// TIA Portal V16 export
// export: Created 2023-05-12T09:02:59.8974602Z, ExportSetting WithDefaults, DisplayName Totally Integrated Automation Portal, DisplayVersion V16 Update 3, DisplayName TIA Portal Version Control Interface, DisplayVersion V16 Update 2, DisplayName TIA Portal Openness, DisplayVersion V16 Update 3, DisplayName SINAMICS Startdrive Advanced, DisplayVersion V16, DisplayName SINAMICS Startdrive G130, G150, S120, S150, SINAMICS MV, S210, DisplayVersion V16, DisplayName SINAMICS Startdrive G110M, G120, G120C, G120D, G120P, DisplayVersion V16, DisplayName STEP 7 Professional, DisplayVersion V16 Update 3, DisplayName STEP 7 Safety, DisplayVersion V16, DisplayName WinCC Advanced, DisplayVersion V16 Update 3
FUNCTION "CIP_LINEA1" : Void   // FC53, LAD
{ S7_Optimized_Access := 'FALSE' }
VERSION : 0.1
// stored: AutoNumber false, IsIECCheckEnabled false, SetENOAutomatically false, UDAEnableTagReadback false
   VAR_TEMP
      AUX_TEM_P1 : S5Time;
      AUX_BOOL_1 : Bool;
   END_VAR
   VAR_TEMP   // added for the SCL form of the ladder/FBD networks
      _w1 : Bool;
      _s5time1 : S5Time;
   END_VAR
BEGIN

REGION Network 1: SOLO EN LIMPIEZA TANQUES
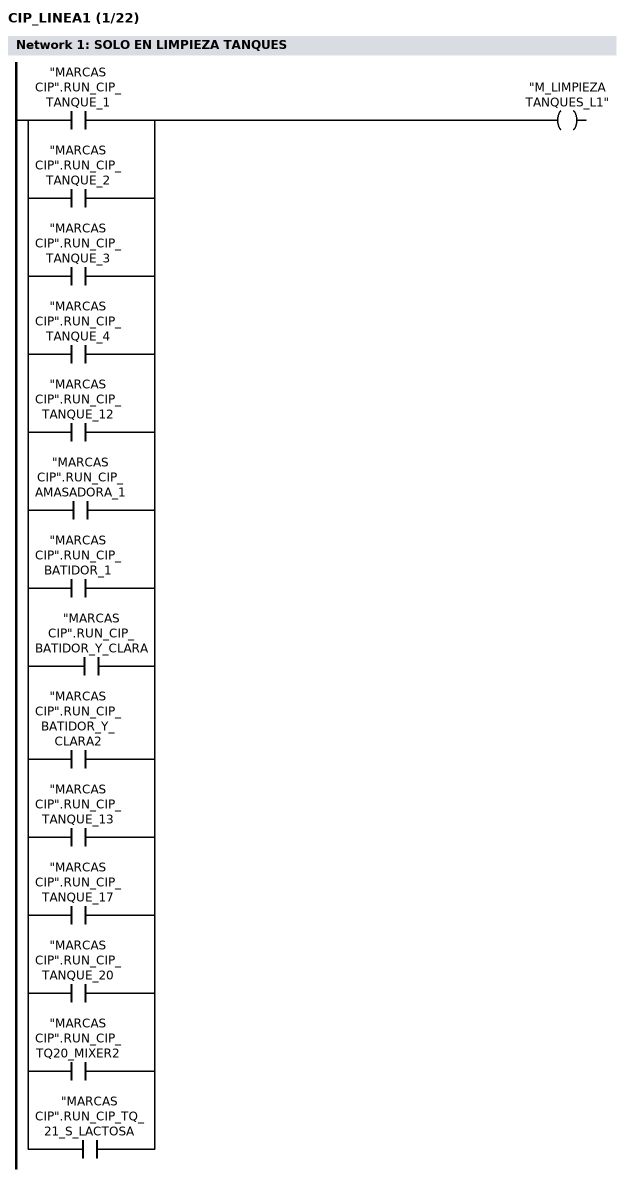
   RUNG wire#powerrail
      Contact( "MARCAS CIP".RUN_CIP_TANQUE_1 )
      wire#w1
      Coil( "M_LIMPIEZA TANQUES_L1" )
   END_RUNG
   RUNG wire#powerrail
      Contact( "MARCAS CIP".RUN_CIP_TANQUE_2 )
   END_RUNG wire#w1
   RUNG wire#powerrail
      Contact( "MARCAS CIP".RUN_CIP_TANQUE_3 )
   END_RUNG wire#w1
   RUNG wire#powerrail
      Contact( "MARCAS CIP".RUN_CIP_TANQUE_4 )
   END_RUNG wire#w1
   RUNG wire#powerrail
      Contact( "MARCAS CIP".RUN_CIP_TANQUE_12 )
   END_RUNG wire#w1
   RUNG wire#powerrail
      Contact( "MARCAS CIP".RUN_CIP_AMASADORA_1 )
   END_RUNG wire#w1
   RUNG wire#powerrail
      Contact( "MARCAS CIP".RUN_CIP_BATIDOR_1 )
   END_RUNG wire#w1
   RUNG wire#powerrail
      Contact( "MARCAS CIP".RUN_CIP_BATIDOR_Y_CLARA )
   END_RUNG wire#w1
   RUNG wire#powerrail
      Contact( "MARCAS CIP".RUN_CIP_BATIDOR_Y_CLARA2 )
   END_RUNG wire#w1
   RUNG wire#powerrail
      Contact( "MARCAS CIP".RUN_CIP_TANQUE_13 )
   END_RUNG wire#w1
   RUNG wire#powerrail
      Contact( "MARCAS CIP".RUN_CIP_TANQUE_17 )
   END_RUNG wire#w1
   RUNG wire#powerrail
      Contact( "MARCAS CIP".RUN_CIP_TANQUE_20 )
   END_RUNG wire#w1
   RUNG wire#powerrail
      Contact( "MARCAS CIP".RUN_CIP_TQ20_MIXER2 )
   END_RUNG wire#w1
   RUNG wire#powerrail
      Contact( "MARCAS CIP".RUN_CIP_TQ_21_S_LACTOSA )
   END_RUNG wire#w1
   // the same network as SCL:
   "M_LIMPIEZA TANQUES_L1" := "MARCAS CIP".RUN_CIP_TANQUE_1 OR "MARCAS CIP".RUN_CIP_TANQUE_2 OR "MARCAS CIP".RUN_CIP_TANQUE_3 OR "MARCAS CIP".RUN_CIP_TANQUE_4 OR "MARCAS CIP".RUN_CIP_TANQUE_12 OR "MARCAS CIP".RUN_CIP_AMASADORA_1 OR "MARCAS CIP".RUN_CIP_BATIDOR_1 OR "MARCAS CIP".RUN_CIP_BATIDOR_Y_CLARA OR "MARCAS CIP".RUN_CIP_BATIDOR_Y_CLARA2 OR "MARCAS CIP".RUN_CIP_TANQUE_13 OR "MARCAS CIP".RUN_CIP_TANQUE_17 OR "MARCAS CIP".RUN_CIP_TANQUE_20 OR "MARCAS CIP".RUN_CIP_TQ20_MIXER2 OR "MARCAS CIP".RUN_CIP_TQ_21_S_LACTOSA;
END_REGION

REGION Network 2: PASO 1 PRIEMER ENJUEGE AGUA RECUPERADA
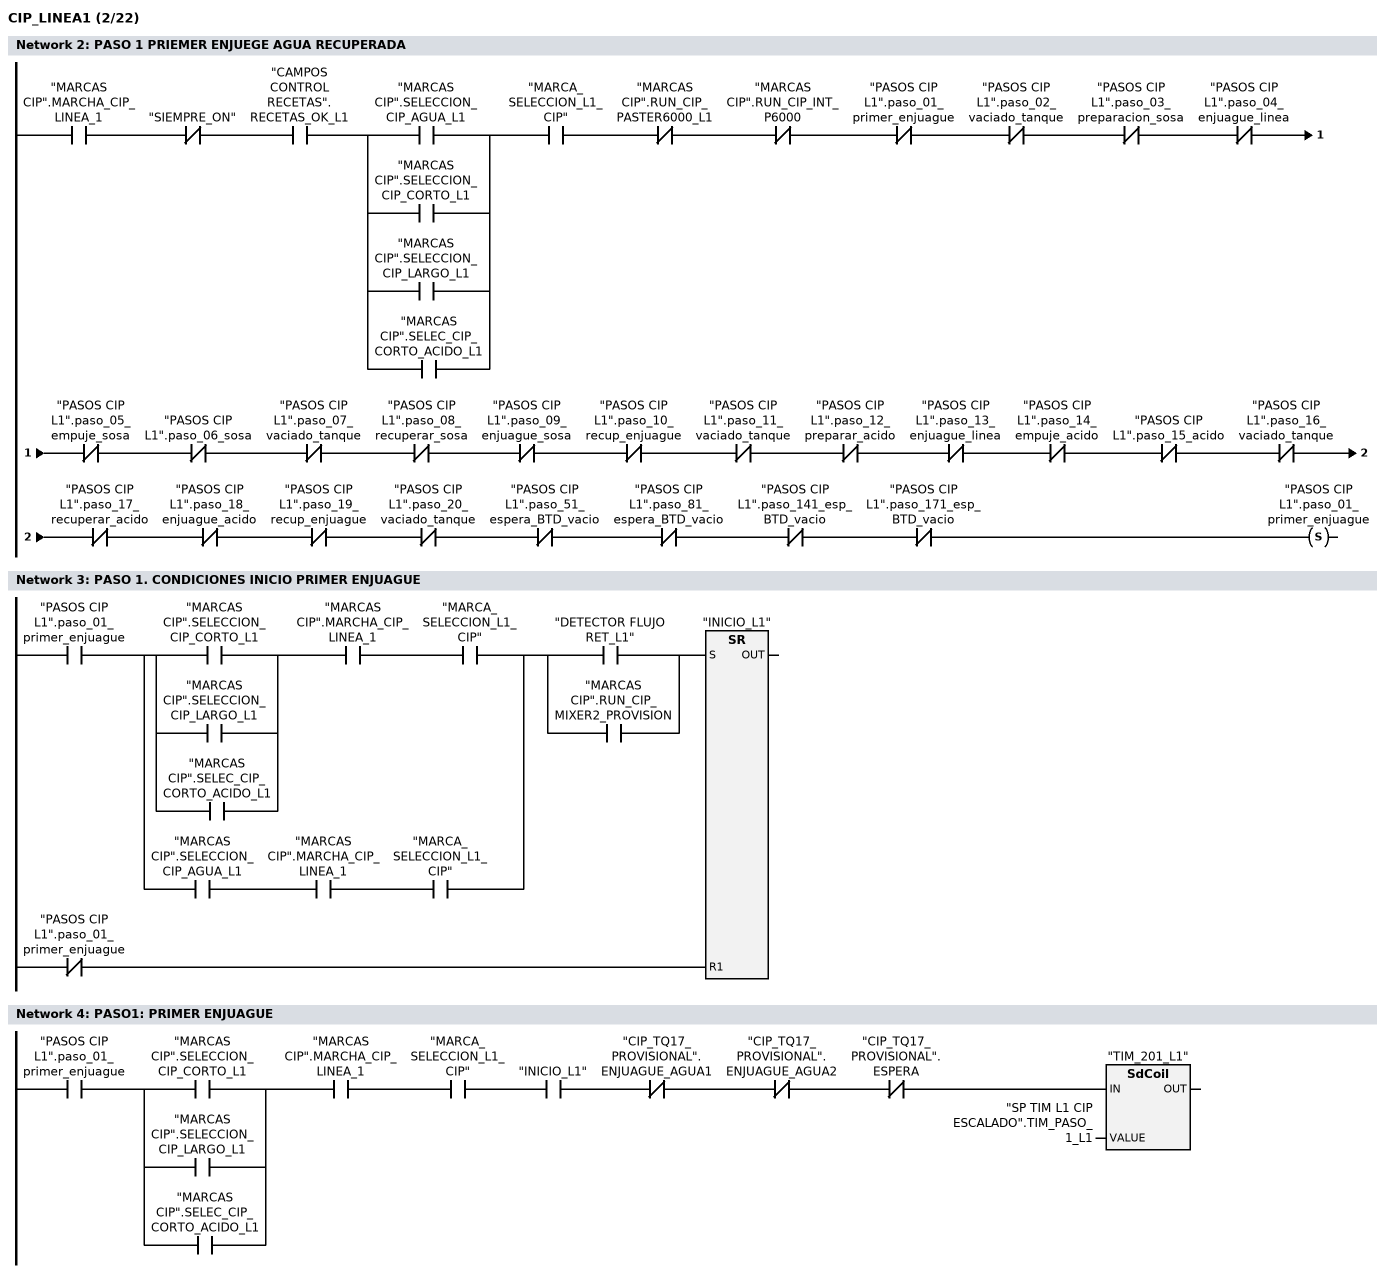
   RUNG wire#powerrail
      Contact( "MARCAS CIP".MARCHA_CIP_LINEA_1 )
      I_Contact( "SIEMPRE_ON" )
      Contact( "CAMPOS CONTROL RECETAS".RECETAS_OK_L1 )
      wire#w1
      Contact( "MARCAS CIP".SELECCION_CIP_AGUA_L1 )
      wire#w2
      Contact( "MARCA_SELECCION_L1_CIP" )
      I_Contact( "MARCAS CIP".RUN_CIP_PASTER6000_L1 )
      I_Contact( "MARCAS CIP".RUN_CIP_INT_P6000 )
      I_Contact( "PASOS CIP L1".paso_01_primer_enjuague )
      I_Contact( "PASOS CIP L1".paso_02_vaciado_tanque )
      I_Contact( "PASOS CIP L1".paso_03_preparacion_sosa )
      I_Contact( "PASOS CIP L1".paso_04_enjuague_linea )
      I_Contact( "PASOS CIP L1".paso_05_empuje_sosa )
      I_Contact( "PASOS CIP L1".paso_06_sosa )
      I_Contact( "PASOS CIP L1".paso_07_vaciado_tanque )
      I_Contact( "PASOS CIP L1".paso_08_recuperar_sosa )
      I_Contact( "PASOS CIP L1".paso_09_enjuague_sosa )
      I_Contact( "PASOS CIP L1".paso_10_recup_enjuague )
      I_Contact( "PASOS CIP L1".paso_11_vaciado_tanque )
      I_Contact( "PASOS CIP L1".paso_12_preparar_acido )
      I_Contact( "PASOS CIP L1".paso_13_enjuague_linea )
      I_Contact( "PASOS CIP L1".paso_14_empuje_acido )
      I_Contact( "PASOS CIP L1".paso_15_acido )
      I_Contact( "PASOS CIP L1".paso_16_vaciado_tanque )
      I_Contact( "PASOS CIP L1".paso_17_recuperar_acido )
      I_Contact( "PASOS CIP L1".paso_18_enjuague_acido )
      I_Contact( "PASOS CIP L1".paso_19_recup_enjuague )
      I_Contact( "PASOS CIP L1".paso_20_vaciado_tanque )
      I_Contact( "PASOS CIP L1".paso_51_espera_BTD_vacio )
      I_Contact( "PASOS CIP L1".paso_81_espera_BTD_vacio )
      I_Contact( "PASOS CIP L1".paso_141_esp_BTD_vacio )
      I_Contact( "PASOS CIP L1".paso_171_esp_BTD_vacio )
      S_Coil( "PASOS CIP L1".paso_01_primer_enjuague )
   END_RUNG
   RUNG wire#w1
      Contact( "MARCAS CIP".SELECCION_CIP_CORTO_L1 )
   END_RUNG wire#w2
   RUNG wire#w1
      Contact( "MARCAS CIP".SELECCION_CIP_LARGO_L1 )
   END_RUNG wire#w2
   RUNG wire#w1
      Contact( "MARCAS CIP".SELEC_CIP_CORTO_ACIDO_L1 )
   END_RUNG wire#w2
   // the same network as SCL:
   IF "MARCAS CIP".MARCHA_CIP_LINEA_1 AND NOT "SIEMPRE_ON" AND "CAMPOS CONTROL RECETAS".RECETAS_OK_L1 AND ("MARCAS CIP".SELECCION_CIP_AGUA_L1 OR "MARCAS CIP".SELECCION_CIP_CORTO_L1 OR "MARCAS CIP".SELECCION_CIP_LARGO_L1 OR "MARCAS CIP".SELEC_CIP_CORTO_ACIDO_L1) AND "MARCA_SELECCION_L1_CIP" AND NOT "MARCAS CIP".RUN_CIP_PASTER6000_L1 AND NOT "MARCAS CIP".RUN_CIP_INT_P6000 AND NOT "PASOS CIP L1".paso_01_primer_enjuague AND NOT "PASOS CIP L1".paso_02_vaciado_tanque AND NOT "PASOS CIP L1".paso_03_preparacion_sosa AND NOT "PASOS CIP L1".paso_04_enjuague_linea AND NOT "PASOS CIP L1".paso_05_empuje_sosa AND NOT "PASOS CIP L1".paso_06_sosa AND NOT "PASOS CIP L1".paso_07_vaciado_tanque AND NOT "PASOS CIP L1".paso_08_recuperar_sosa AND NOT "PASOS CIP L1".paso_09_enjuague_sosa AND NOT "PASOS CIP L1".paso_10_recup_enjuague AND NOT "PASOS CIP L1".paso_11_vaciado_tanque AND NOT "PASOS CIP L1".paso_12_preparar_acido AND NOT "PASOS CIP L1".paso_13_enjuague_linea AND NOT "PASOS CIP L1".paso_14_empuje_acido AND NOT "PASOS CIP L1".paso_15_acido AND NOT "PASOS CIP L1".paso_16_vaciado_tanque AND NOT "PASOS CIP L1".paso_17_recuperar_acido AND NOT "PASOS CIP L1".paso_18_enjuague_acido AND NOT "PASOS CIP L1".paso_19_recup_enjuague AND NOT "PASOS CIP L1".paso_20_vaciado_tanque AND NOT "PASOS CIP L1".paso_51_espera_BTD_vacio AND NOT "PASOS CIP L1".paso_81_espera_BTD_vacio AND NOT "PASOS CIP L1".paso_141_esp_BTD_vacio AND NOT "PASOS CIP L1".paso_171_esp_BTD_vacio THEN
       "PASOS CIP L1".paso_01_primer_enjuague := TRUE;
   END_IF;
END_REGION

REGION Network 3: PASO 1. CONDICIONES INICIO PRIMER ENJUAGUE
   RUNG wire#powerrail
      Contact( "PASOS CIP L1".paso_01_primer_enjuague )
      wire#w1
      Contact( "MARCAS CIP".SELECCION_CIP_CORTO_L1 )
      wire#w2
      Contact( "MARCAS CIP".MARCHA_CIP_LINEA_1 )
      Contact( "MARCA_SELECCION_L1_CIP" )
      wire#w3
      Contact( "DETECTOR FLUJO RET_L1" )
      wire#w4
      S_SR(operand := "INICIO_L1", r1 := wire#w5)
   END_RUNG
   RUNG wire#w1
      Contact( "MARCAS CIP".SELECCION_CIP_LARGO_L1 )
   END_RUNG wire#w2
   RUNG wire#w1
      Contact( "MARCAS CIP".SELEC_CIP_CORTO_ACIDO_L1 )
   END_RUNG wire#w2
   RUNG wire#w1
      Contact( "MARCAS CIP".SELECCION_CIP_AGUA_L1 )
      Contact( "MARCAS CIP".MARCHA_CIP_LINEA_1 )
      Contact( "MARCA_SELECCION_L1_CIP" )
   END_RUNG wire#w3
   RUNG wire#w3
      Contact( "MARCAS CIP".RUN_CIP_MIXER2_PROVISION )
   END_RUNG wire#w4
   RUNG wire#powerrail
      I_Contact( "PASOS CIP L1".paso_01_primer_enjuague )
   END_RUNG wire#w5
   // the same network as SCL:
   IF "PASOS CIP L1".paso_01_primer_enjuague AND ((("MARCAS CIP".SELECCION_CIP_CORTO_L1 OR "MARCAS CIP".SELECCION_CIP_LARGO_L1 OR "MARCAS CIP".SELEC_CIP_CORTO_ACIDO_L1) AND "MARCAS CIP".MARCHA_CIP_LINEA_1 AND "MARCA_SELECCION_L1_CIP") OR ("MARCAS CIP".SELECCION_CIP_AGUA_L1 AND "MARCAS CIP".MARCHA_CIP_LINEA_1 AND "MARCA_SELECCION_L1_CIP")) AND ("DETECTOR FLUJO RET_L1" OR "MARCAS CIP".RUN_CIP_MIXER2_PROVISION) THEN
       "INICIO_L1" := TRUE;   // SR flip-flop
   END_IF;
   IF NOT "PASOS CIP L1".paso_01_primer_enjuague THEN "INICIO_L1" := FALSE; END_IF;
END_REGION

REGION Network 4: PASO1: PRIMER ENJUAGUE
   // no SCL statement known for SdCoil: written as a call
   SdCoil(value := "SP TIM L1 CIP ESCALADO".TIM_PASO_1_L1,
          operand := "TIM_201_L1",
          in := "PASOS CIP L1".paso_01_primer_enjuague AND ("MARCAS CIP".SELECCION_CIP_CORTO_L1 OR "MARCAS CIP".SELECCION_CIP_LARGO_L1 OR "MARCAS CIP".SELEC_CIP_CORTO_ACIDO_L1) AND "MARCAS CIP".MARCHA_CIP_LINEA_1 AND "MARCA_SELECCION_L1_CIP" AND "INICIO_L1" AND NOT "CIP_TQ17_PROVISIONAL".ENJUAGUE_AGUA1 AND NOT "CIP_TQ17_PROVISIONAL".ENJUAGUE_AGUA2 AND NOT "CIP_TQ17_PROVISIONAL".ESPERA);
END_REGION

REGION Network 5: PASO 2: VACIADO TANQUE (SOLO BOMBA RETORNO CIP)
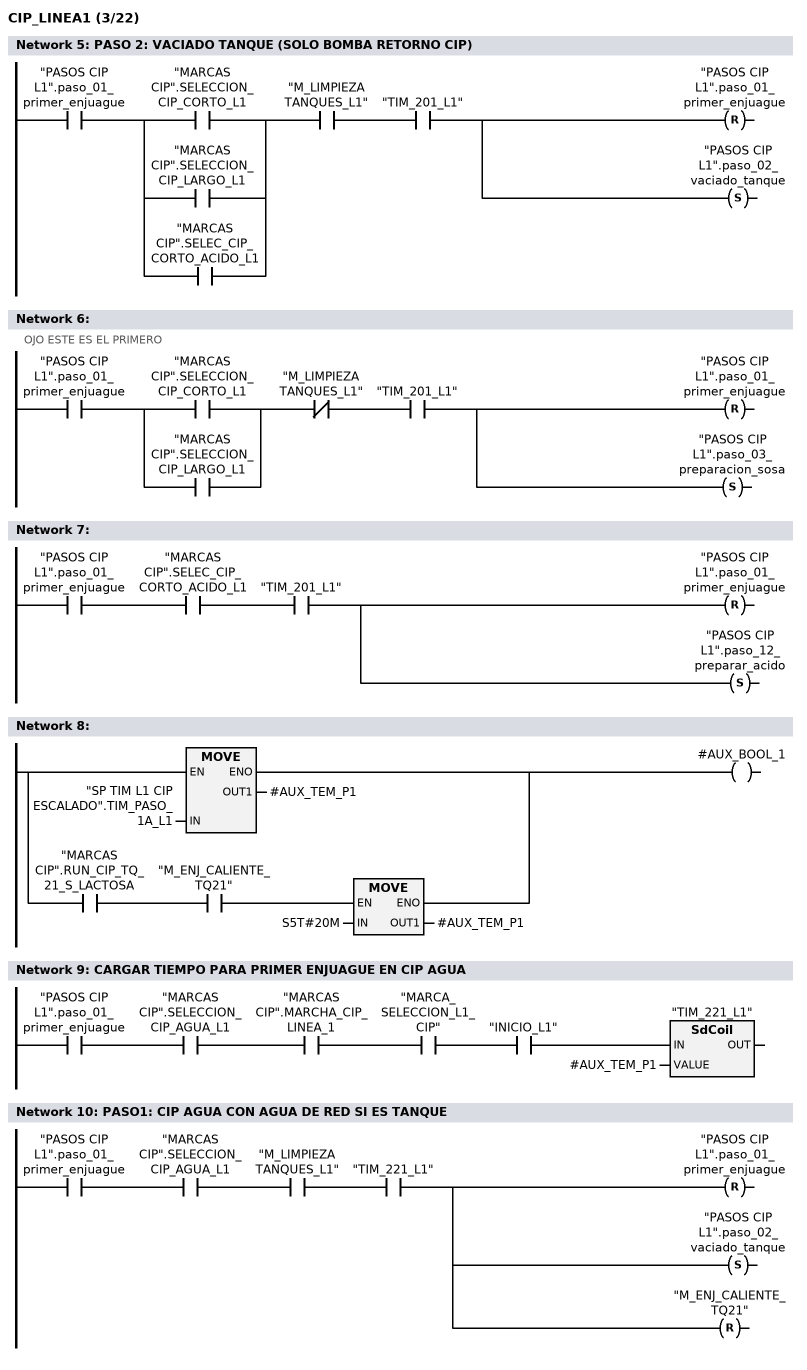
   RUNG wire#powerrail
      Contact( "PASOS CIP L1".paso_01_primer_enjuague )
      wire#w1
      Contact( "MARCAS CIP".SELECCION_CIP_CORTO_L1 )
      wire#w2
      Contact( "M_LIMPIEZA TANQUES_L1" )
      Contact( "TIM_201_L1" )
      wire#w3
      R_Coil( "PASOS CIP L1".paso_01_primer_enjuague )
   END_RUNG
   RUNG wire#w1
      Contact( "MARCAS CIP".SELECCION_CIP_LARGO_L1 )
   END_RUNG wire#w2
   RUNG wire#w1
      Contact( "MARCAS CIP".SELEC_CIP_CORTO_ACIDO_L1 )
   END_RUNG wire#w2
   RUNG wire#w3
      S_Coil( "PASOS CIP L1".paso_02_vaciado_tanque )
   END_RUNG
   // the same network as SCL:
   #_w1 := "PASOS CIP L1".paso_01_primer_enjuague AND ("MARCAS CIP".SELECCION_CIP_CORTO_L1 OR "MARCAS CIP".SELECCION_CIP_LARGO_L1 OR "MARCAS CIP".SELEC_CIP_CORTO_ACIDO_L1) AND "M_LIMPIEZA TANQUES_L1" AND "TIM_201_L1";
   IF #_w1 THEN
       "PASOS CIP L1".paso_01_primer_enjuague := FALSE;
       "PASOS CIP L1".paso_02_vaciado_tanque := TRUE;
   END_IF;
END_REGION

REGION Network 6
   // OJO ESTE ES EL PRIMERO
   RUNG wire#powerrail
      Contact( "PASOS CIP L1".paso_01_primer_enjuague )
      wire#w1
      Contact( "MARCAS CIP".SELECCION_CIP_CORTO_L1 )
      wire#w2
      I_Contact( "M_LIMPIEZA TANQUES_L1" )
      Contact( "TIM_201_L1" )
      wire#w3
      R_Coil( "PASOS CIP L1".paso_01_primer_enjuague )
   END_RUNG
   RUNG wire#w1
      Contact( "MARCAS CIP".SELECCION_CIP_LARGO_L1 )
   END_RUNG wire#w2
   RUNG wire#w3
      S_Coil( "PASOS CIP L1".paso_03_preparacion_sosa )
   END_RUNG
   // the same network as SCL:
   #_w1 := "PASOS CIP L1".paso_01_primer_enjuague AND ("MARCAS CIP".SELECCION_CIP_CORTO_L1 OR "MARCAS CIP".SELECCION_CIP_LARGO_L1) AND NOT "M_LIMPIEZA TANQUES_L1" AND "TIM_201_L1";
   IF #_w1 THEN
       "PASOS CIP L1".paso_01_primer_enjuague := FALSE;
       "PASOS CIP L1".paso_03_preparacion_sosa := TRUE;
   END_IF;
END_REGION

REGION Network 7
   RUNG wire#powerrail
      Contact( "PASOS CIP L1".paso_01_primer_enjuague )
      Contact( "MARCAS CIP".SELEC_CIP_CORTO_ACIDO_L1 )
      Contact( "TIM_201_L1" )
      wire#w1
      R_Coil( "PASOS CIP L1".paso_01_primer_enjuague )
   END_RUNG
   RUNG wire#w1
      S_Coil( "PASOS CIP L1".paso_12_preparar_acido )
   END_RUNG
   // the same network as SCL:
   #_w1 := "PASOS CIP L1".paso_01_primer_enjuague AND "MARCAS CIP".SELEC_CIP_CORTO_ACIDO_L1 AND "TIM_201_L1";
   IF #_w1 THEN
       "PASOS CIP L1".paso_01_primer_enjuague := FALSE;
       "PASOS CIP L1".paso_12_preparar_acido := TRUE;
   END_IF;
END_REGION

REGION Network 8
   RUNG wire#powerrail
      { S7_GenerateENO := "TRUE" } Move(in := "SP TIM L1 CIP ESCALADO".TIM_PASO_1A_L1, out1 => #AUX_TEM_P1)
      wire#w1
      Coil( #AUX_BOOL_1 )
   END_RUNG
   RUNG wire#powerrail
      Contact( "MARCAS CIP".RUN_CIP_TQ_21_S_LACTOSA )
      Contact( "M_ENJ_CALIENTE_TQ21" )
      { S7_GenerateENO := "TRUE" } Move(in := S5T#20M, out1 => #AUX_TEM_P1)
   END_RUNG wire#w1
   // the same network as SCL:
   // ENO of a box is taken as its EN; it also drops when the box reports an error
   #AUX_TEM_P1 := "SP TIM L1 CIP ESCALADO".TIM_PASO_1A_L1;
   #_w1 := "MARCAS CIP".RUN_CIP_TQ_21_S_LACTOSA AND "M_ENJ_CALIENTE_TQ21";
   IF #_w1 THEN #AUX_TEM_P1 := S5T#20M; END_IF;
   #AUX_BOOL_1 := TRUE OR #_w1;
END_REGION

REGION Network 9: CARGAR TIEMPO PARA PRIMER ENJUAGUE EN CIP AGUA
   // no SCL statement known for SdCoil: written as a call
   SdCoil(value := #AUX_TEM_P1,
          operand := "TIM_221_L1",
          in := "PASOS CIP L1".paso_01_primer_enjuague AND "MARCAS CIP".SELECCION_CIP_AGUA_L1 AND "MARCAS CIP".MARCHA_CIP_LINEA_1 AND "MARCA_SELECCION_L1_CIP" AND "INICIO_L1");
END_REGION

REGION Network 10: PASO1: CIP AGUA CON AGUA DE RED SI ES TANQUE
   RUNG wire#powerrail
      Contact( "PASOS CIP L1".paso_01_primer_enjuague )
      Contact( "MARCAS CIP".SELECCION_CIP_AGUA_L1 )
      Contact( "M_LIMPIEZA TANQUES_L1" )
      Contact( "TIM_221_L1" )
      wire#w1
      R_Coil( "PASOS CIP L1".paso_01_primer_enjuague )
   END_RUNG
   RUNG wire#w1
      S_Coil( "PASOS CIP L1".paso_02_vaciado_tanque )
   END_RUNG
   RUNG wire#w1
      R_Coil( "M_ENJ_CALIENTE_TQ21" )
   END_RUNG
   // the same network as SCL:
   #_w1 := "PASOS CIP L1".paso_01_primer_enjuague AND "MARCAS CIP".SELECCION_CIP_AGUA_L1 AND "M_LIMPIEZA TANQUES_L1" AND "TIM_221_L1";
   IF #_w1 THEN
       "PASOS CIP L1".paso_01_primer_enjuague := FALSE;
       "PASOS CIP L1".paso_02_vaciado_tanque := TRUE;
       "M_ENJ_CALIENTE_TQ21" := FALSE;
   END_IF;
END_REGION

REGION Network 11: PASO1: CIP AGUA CON AGUA DE RED SI ES LINEA
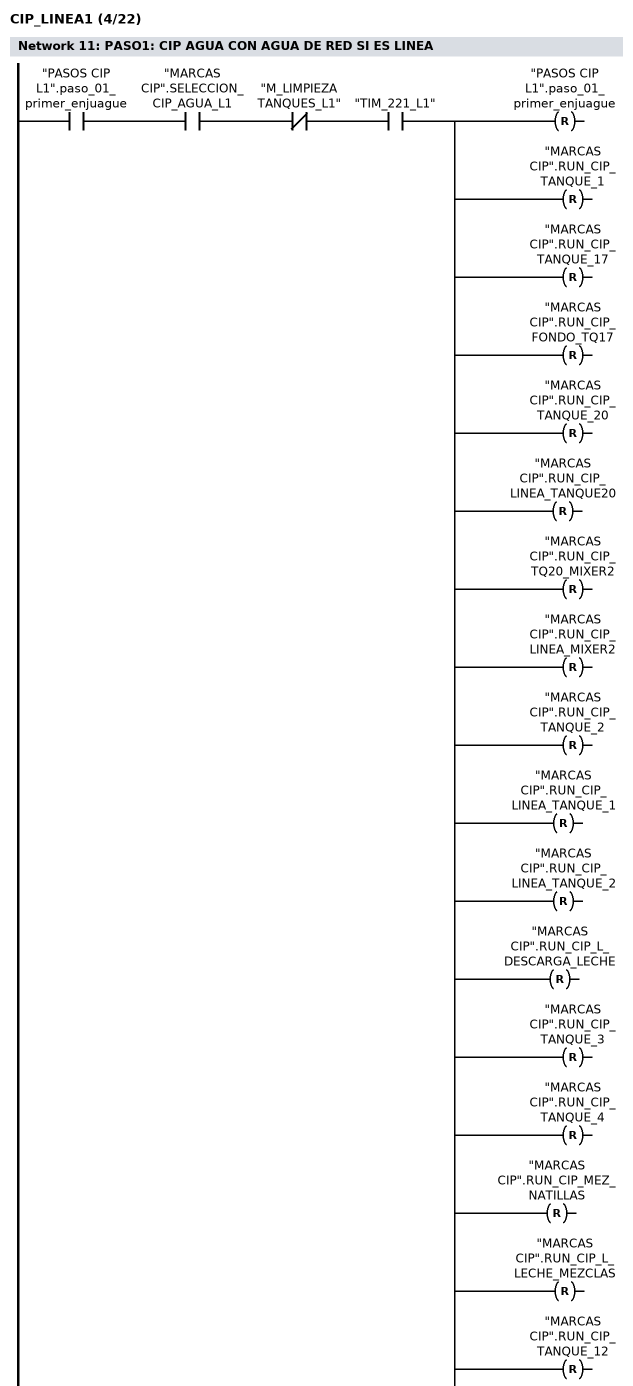
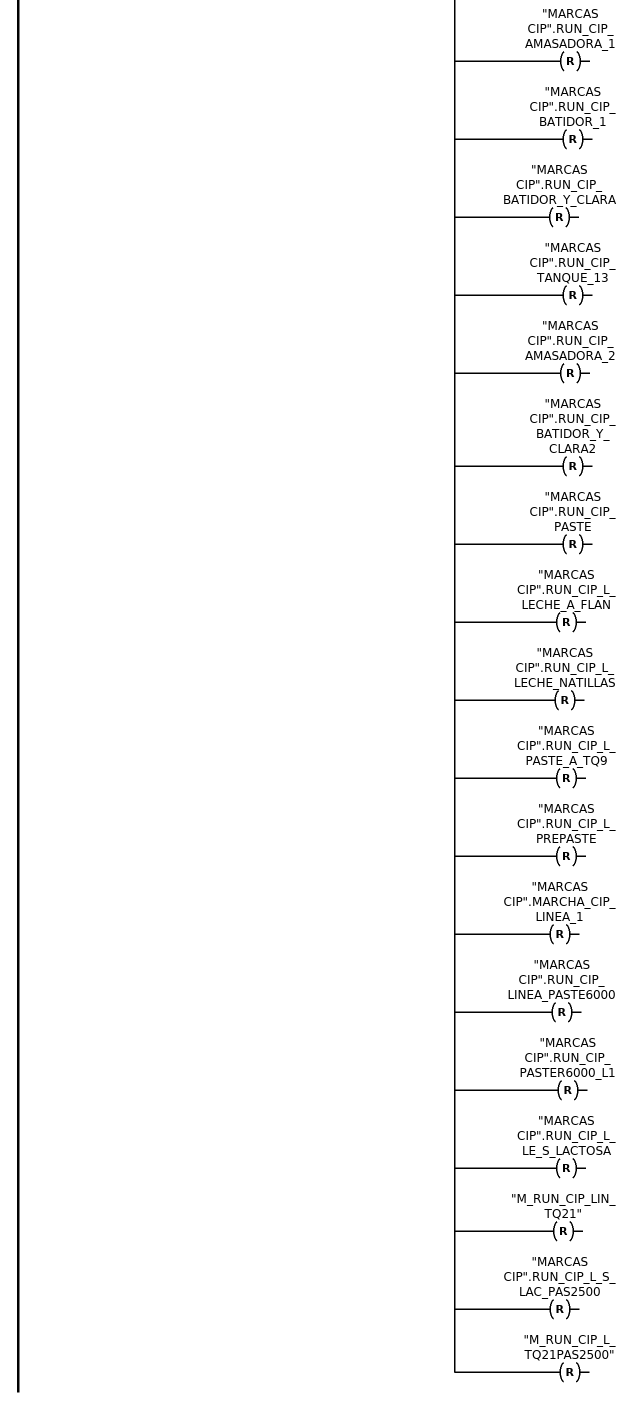
   RUNG wire#powerrail
      Contact( "PASOS CIP L1".paso_01_primer_enjuague )
      Contact( "MARCAS CIP".SELECCION_CIP_AGUA_L1 )
      I_Contact( "M_LIMPIEZA TANQUES_L1" )
      Contact( "TIM_221_L1" )
      wire#w1
      R_Coil( "PASOS CIP L1".paso_01_primer_enjuague )
   END_RUNG
   RUNG wire#w1
      R_Coil( "MARCAS CIP".RUN_CIP_TANQUE_1 )
   END_RUNG
   RUNG wire#w1
      R_Coil( "MARCAS CIP".RUN_CIP_TANQUE_17 )
   END_RUNG
   RUNG wire#w1
      R_Coil( "MARCAS CIP".RUN_CIP_FONDO_TQ17 )
   END_RUNG
   RUNG wire#w1
      R_Coil( "MARCAS CIP".RUN_CIP_TANQUE_20 )
   END_RUNG
   RUNG wire#w1
      R_Coil( "MARCAS CIP".RUN_CIP_LINEA_TANQUE20 )
   END_RUNG
   RUNG wire#w1
      R_Coil( "MARCAS CIP".RUN_CIP_TQ20_MIXER2 )
   END_RUNG
   RUNG wire#w1
      R_Coil( "MARCAS CIP".RUN_CIP_LINEA_MIXER2 )
   END_RUNG
   RUNG wire#w1
      R_Coil( "MARCAS CIP".RUN_CIP_TANQUE_2 )
   END_RUNG
   RUNG wire#w1
      R_Coil( "MARCAS CIP".RUN_CIP_LINEA_TANQUE_1 )
   END_RUNG
   RUNG wire#w1
      R_Coil( "MARCAS CIP".RUN_CIP_LINEA_TANQUE_2 )
   END_RUNG
   RUNG wire#w1
      R_Coil( "MARCAS CIP".RUN_CIP_L_DESCARGA_LECHE )
   END_RUNG
   RUNG wire#w1
      R_Coil( "MARCAS CIP".RUN_CIP_TANQUE_3 )
   END_RUNG
   RUNG wire#w1
      R_Coil( "MARCAS CIP".RUN_CIP_TANQUE_4 )
   END_RUNG
   RUNG wire#w1
      R_Coil( "MARCAS CIP".RUN_CIP_MEZ_NATILLAS )
   END_RUNG
   RUNG wire#w1
      R_Coil( "MARCAS CIP".RUN_CIP_L_LECHE_MEZCLAS )
   END_RUNG
   RUNG wire#w1
      R_Coil( "MARCAS CIP".RUN_CIP_TANQUE_12 )
   END_RUNG
   RUNG wire#w1
      R_Coil( "MARCAS CIP".RUN_CIP_AMASADORA_1 )
   END_RUNG
   RUNG wire#w1
      R_Coil( "MARCAS CIP".RUN_CIP_BATIDOR_1 )
   END_RUNG
   RUNG wire#w1
      R_Coil( "MARCAS CIP".RUN_CIP_BATIDOR_Y_CLARA )
   END_RUNG
   RUNG wire#w1
      R_Coil( "MARCAS CIP".RUN_CIP_TANQUE_13 )
   END_RUNG
   RUNG wire#w1
      R_Coil( "MARCAS CIP".RUN_CIP_AMASADORA_2 )
   END_RUNG
   RUNG wire#w1
      R_Coil( "MARCAS CIP".RUN_CIP_BATIDOR_Y_CLARA2 )
   END_RUNG
   RUNG wire#w1
      R_Coil( "MARCAS CIP".RUN_CIP_PASTE )
   END_RUNG
   RUNG wire#w1
      R_Coil( "MARCAS CIP".RUN_CIP_L_LECHE_A_FLAN )
   END_RUNG
   RUNG wire#w1
      R_Coil( "MARCAS CIP".RUN_CIP_L_LECHE_NATILLAS )
   END_RUNG
   RUNG wire#w1
      R_Coil( "MARCAS CIP".RUN_CIP_L_PASTE_A_TQ9 )
   END_RUNG
   RUNG wire#w1
      R_Coil( "MARCAS CIP".RUN_CIP_L_PREPASTE )
   END_RUNG
   RUNG wire#w1
      R_Coil( "MARCAS CIP".MARCHA_CIP_LINEA_1 )
   END_RUNG
   RUNG wire#w1
      R_Coil( "MARCAS CIP".RUN_CIP_LINEA_PASTE6000 )
   END_RUNG
   RUNG wire#w1
      R_Coil( "MARCAS CIP".RUN_CIP_PASTER6000_L1 )
   END_RUNG
   RUNG wire#w1
      R_Coil( "MARCAS CIP".RUN_CIP_L_LE_S_LACTOSA )
   END_RUNG
   RUNG wire#w1
      R_Coil( "M_RUN_CIP_LIN_TQ21" )
   END_RUNG
   RUNG wire#w1
      R_Coil( "MARCAS CIP".RUN_CIP_L_S_LAC_PAS2500 )
   END_RUNG
   RUNG wire#w1
      R_Coil( "M_RUN_CIP_L_TQ21PAS2500" )
   END_RUNG
   // the same network as SCL:
   #_w1 := "PASOS CIP L1".paso_01_primer_enjuague AND "MARCAS CIP".SELECCION_CIP_AGUA_L1 AND NOT "M_LIMPIEZA TANQUES_L1" AND "TIM_221_L1";
   IF #_w1 THEN
       "PASOS CIP L1".paso_01_primer_enjuague := FALSE;
       "MARCAS CIP".RUN_CIP_TANQUE_1 := FALSE;
       "MARCAS CIP".RUN_CIP_TANQUE_17 := FALSE;
       "MARCAS CIP".RUN_CIP_FONDO_TQ17 := FALSE;
       "MARCAS CIP".RUN_CIP_TANQUE_20 := FALSE;
       "MARCAS CIP".RUN_CIP_LINEA_TANQUE20 := FALSE;
       "MARCAS CIP".RUN_CIP_TQ20_MIXER2 := FALSE;
       "MARCAS CIP".RUN_CIP_LINEA_MIXER2 := FALSE;
       "MARCAS CIP".RUN_CIP_TANQUE_2 := FALSE;
       "MARCAS CIP".RUN_CIP_LINEA_TANQUE_1 := FALSE;
       "MARCAS CIP".RUN_CIP_LINEA_TANQUE_2 := FALSE;
       "MARCAS CIP".RUN_CIP_L_DESCARGA_LECHE := FALSE;
       "MARCAS CIP".RUN_CIP_TANQUE_3 := FALSE;
       "MARCAS CIP".RUN_CIP_TANQUE_4 := FALSE;
       "MARCAS CIP".RUN_CIP_MEZ_NATILLAS := FALSE;
       "MARCAS CIP".RUN_CIP_L_LECHE_MEZCLAS := FALSE;
       "MARCAS CIP".RUN_CIP_TANQUE_12 := FALSE;
       "MARCAS CIP".RUN_CIP_AMASADORA_1 := FALSE;
       "MARCAS CIP".RUN_CIP_BATIDOR_1 := FALSE;
       "MARCAS CIP".RUN_CIP_BATIDOR_Y_CLARA := FALSE;
       "MARCAS CIP".RUN_CIP_TANQUE_13 := FALSE;
       "MARCAS CIP".RUN_CIP_AMASADORA_2 := FALSE;
       "MARCAS CIP".RUN_CIP_BATIDOR_Y_CLARA2 := FALSE;
       "MARCAS CIP".RUN_CIP_PASTE := FALSE;
       "MARCAS CIP".RUN_CIP_L_LECHE_A_FLAN := FALSE;
       "MARCAS CIP".RUN_CIP_L_LECHE_NATILLAS := FALSE;
       "MARCAS CIP".RUN_CIP_L_PASTE_A_TQ9 := FALSE;
       "MARCAS CIP".RUN_CIP_L_PREPASTE := FALSE;
       "MARCAS CIP".MARCHA_CIP_LINEA_1 := FALSE;
       "MARCAS CIP".RUN_CIP_LINEA_PASTE6000 := FALSE;
       "MARCAS CIP".RUN_CIP_PASTER6000_L1 := FALSE;
       "MARCAS CIP".RUN_CIP_L_LE_S_LACTOSA := FALSE;
       "M_RUN_CIP_LIN_TQ21" := FALSE;
       "MARCAS CIP".RUN_CIP_L_S_LAC_PAS2500 := FALSE;
       "M_RUN_CIP_L_TQ21PAS2500" := FALSE;
   END_IF;
END_REGION

REGION Network 12
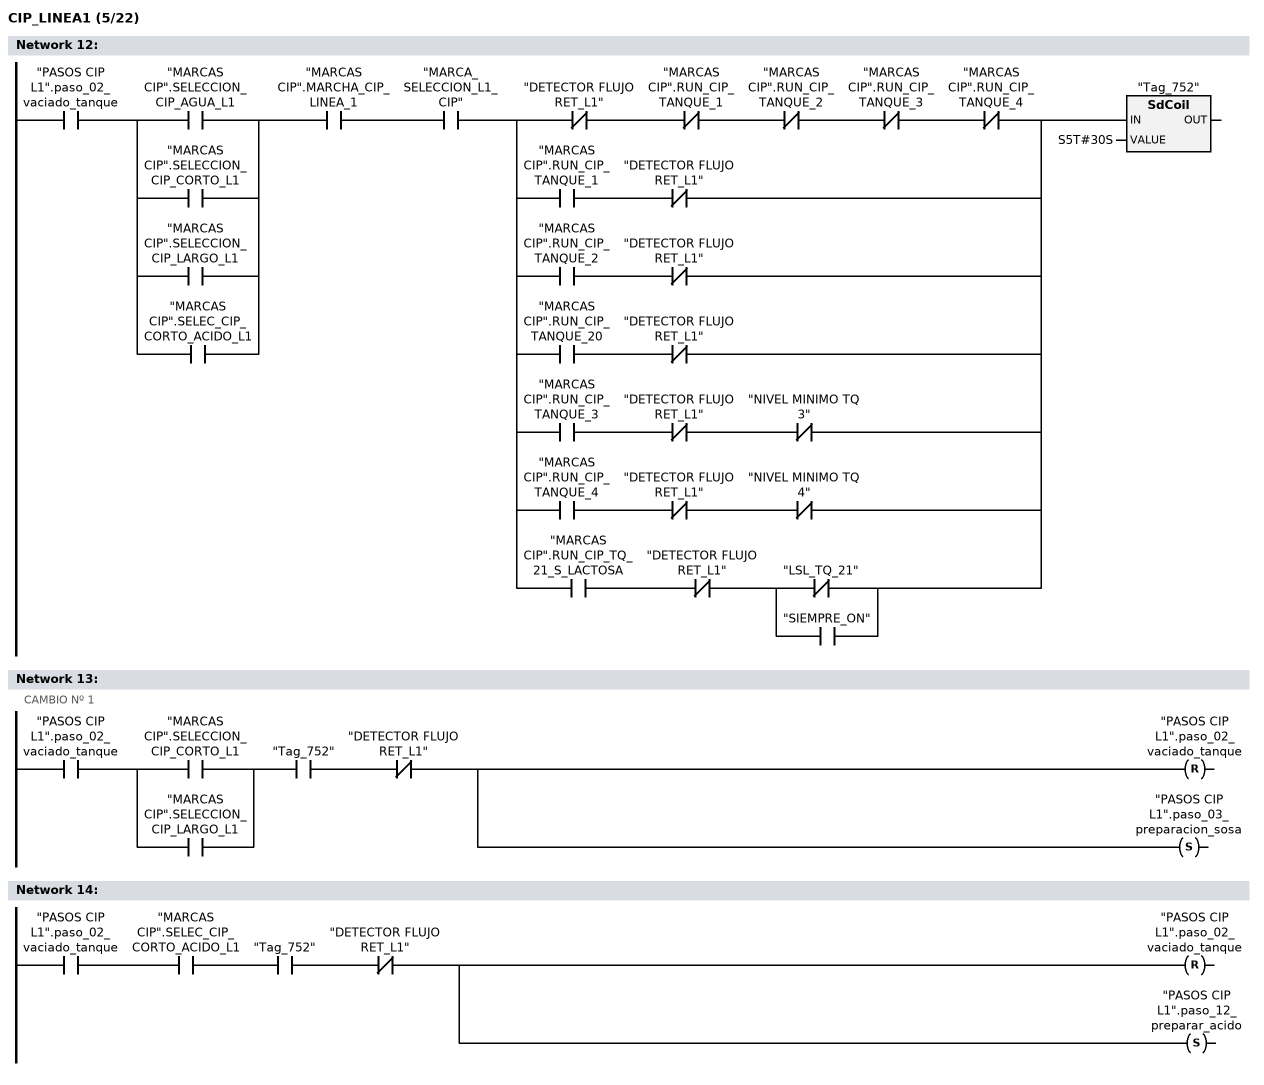
   // no SCL statement known for SdCoil: written as a call
   SdCoil(value := S5T#30S,
          in := "PASOS CIP L1".paso_02_vaciado_tanque AND ("MARCAS CIP".SELECCION_CIP_AGUA_L1 OR "MARCAS CIP".SELECCION_CIP_CORTO_L1 OR "MARCAS CIP".SELECCION_CIP_LARGO_L1 OR "MARCAS CIP".SELEC_CIP_CORTO_ACIDO_L1) AND "MARCAS CIP".MARCHA_CIP_LINEA_1 AND "MARCA_SELECCION_L1_CIP" AND ((NOT "DETECTOR FLUJO RET_L1" AND NOT "MARCAS CIP".RUN_CIP_TANQUE_1 AND NOT "MARCAS CIP".RUN_CIP_TANQUE_2 AND NOT "MARCAS CIP".RUN_CIP_TANQUE_3 AND NOT "MARCAS CIP".RUN_CIP_TANQUE_4) OR ("MARCAS CIP".RUN_CIP_TANQUE_1 AND NOT "DETECTOR FLUJO RET_L1") OR ("MARCAS CIP".RUN_CIP_TANQUE_2 AND NOT "DETECTOR FLUJO RET_L1") OR ("MARCAS CIP".RUN_CIP_TANQUE_20 AND NOT "DETECTOR FLUJO RET_L1") OR ("MARCAS CIP".RUN_CIP_TANQUE_3 AND NOT "DETECTOR FLUJO RET_L1" AND NOT "NIVEL MINIMO TQ 3") OR ("MARCAS CIP".RUN_CIP_TANQUE_4 AND NOT "DETECTOR FLUJO RET_L1" AND NOT "NIVEL MINIMO TQ 4") OR ("MARCAS CIP".RUN_CIP_TQ_21_S_LACTOSA AND NOT "DETECTOR FLUJO RET_L1" AND (NOT "LSL_TQ_21" OR "SIEMPRE_ON"))),
          operand := "Tag_752");
END_REGION

REGION Network 13
   // CAMBIO Nº 1
   RUNG wire#powerrail
      Contact( "PASOS CIP L1".paso_02_vaciado_tanque )
      wire#w1
      Contact( "MARCAS CIP".SELECCION_CIP_CORTO_L1 )
      wire#w2
      Contact( "Tag_752" )
      I_Contact( "DETECTOR FLUJO RET_L1" )
      wire#w3
      R_Coil( "PASOS CIP L1".paso_02_vaciado_tanque )
   END_RUNG
   RUNG wire#w1
      Contact( "MARCAS CIP".SELECCION_CIP_LARGO_L1 )
   END_RUNG wire#w2
   RUNG wire#w3
      S_Coil( "PASOS CIP L1".paso_03_preparacion_sosa )
   END_RUNG
   // the same network as SCL:
   #_w1 := "PASOS CIP L1".paso_02_vaciado_tanque AND ("MARCAS CIP".SELECCION_CIP_CORTO_L1 OR "MARCAS CIP".SELECCION_CIP_LARGO_L1) AND "Tag_752" AND NOT "DETECTOR FLUJO RET_L1";
   IF #_w1 THEN
       "PASOS CIP L1".paso_02_vaciado_tanque := FALSE;
       "PASOS CIP L1".paso_03_preparacion_sosa := TRUE;
   END_IF;
END_REGION

REGION Network 14
   RUNG wire#powerrail
      Contact( "PASOS CIP L1".paso_02_vaciado_tanque )
      Contact( "MARCAS CIP".SELEC_CIP_CORTO_ACIDO_L1 )
      Contact( "Tag_752" )
      I_Contact( "DETECTOR FLUJO RET_L1" )
      wire#w1
      R_Coil( "PASOS CIP L1".paso_02_vaciado_tanque )
   END_RUNG
   RUNG wire#w1
      S_Coil( "PASOS CIP L1".paso_12_preparar_acido )
   END_RUNG
   // the same network as SCL:
   #_w1 := "PASOS CIP L1".paso_02_vaciado_tanque AND "MARCAS CIP".SELEC_CIP_CORTO_ACIDO_L1 AND "Tag_752" AND NOT "DETECTOR FLUJO RET_L1";
   IF #_w1 THEN
       "PASOS CIP L1".paso_02_vaciado_tanque := FALSE;
       "PASOS CIP L1".paso_12_preparar_acido := TRUE;
   END_IF;
END_REGION

REGION Network 15
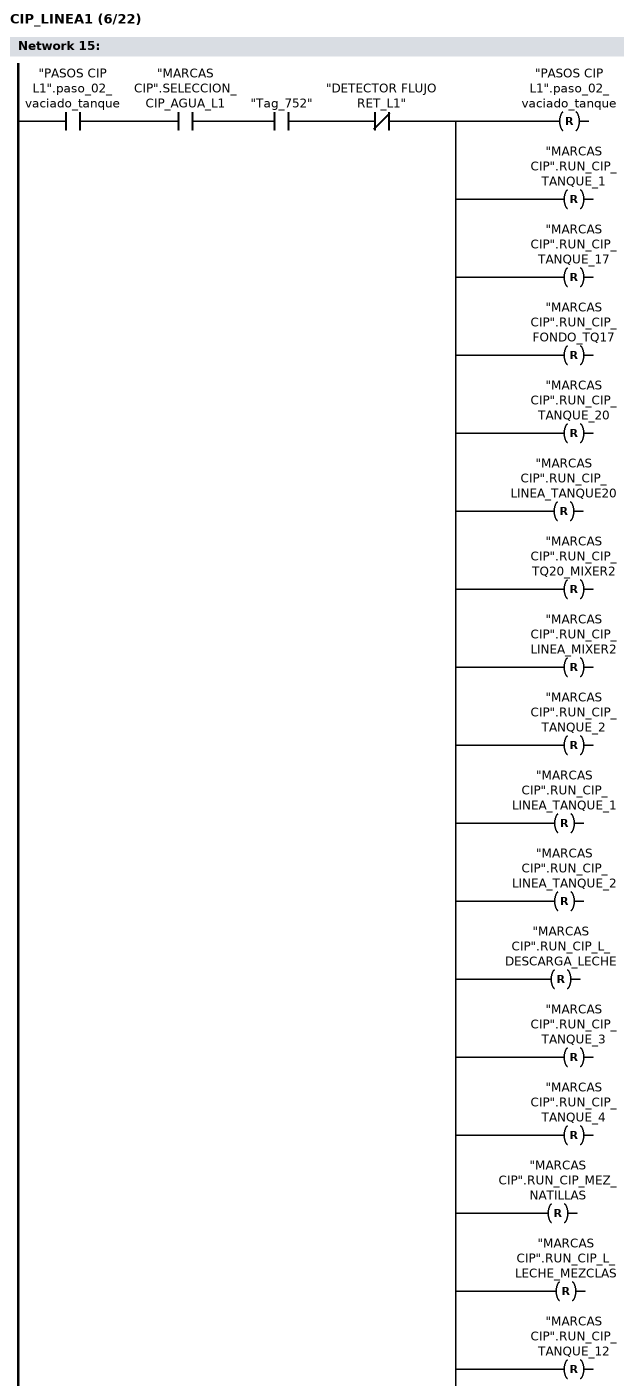
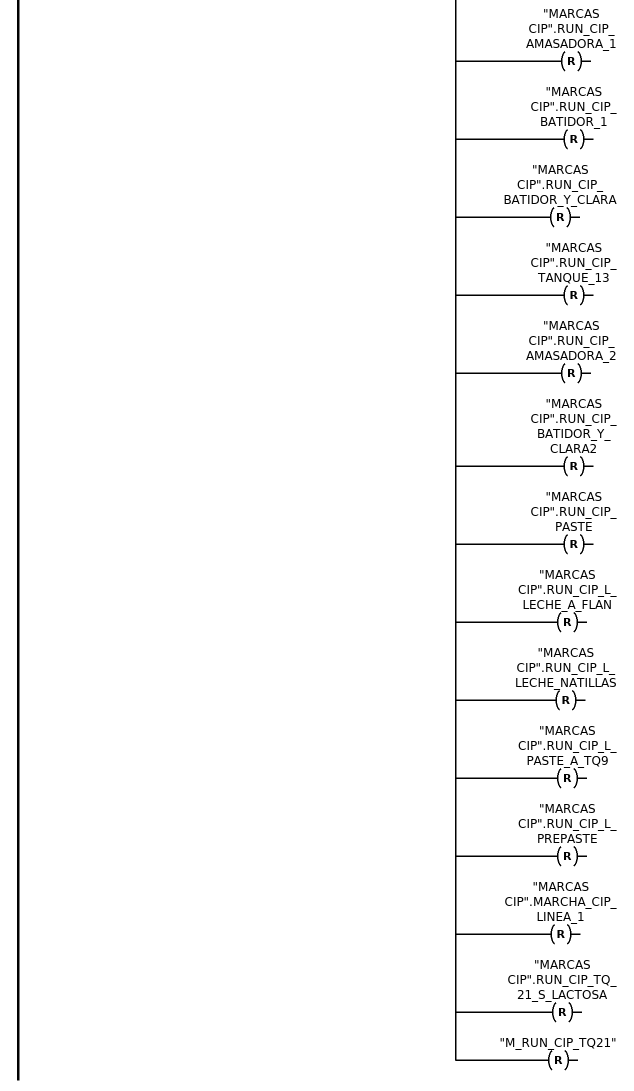
   RUNG wire#powerrail
      Contact( "PASOS CIP L1".paso_02_vaciado_tanque )
      Contact( "MARCAS CIP".SELECCION_CIP_AGUA_L1 )
      Contact( "Tag_752" )
      I_Contact( "DETECTOR FLUJO RET_L1" )
      wire#w1
      R_Coil( "PASOS CIP L1".paso_02_vaciado_tanque )
   END_RUNG
   RUNG wire#w1
      R_Coil( "MARCAS CIP".RUN_CIP_TANQUE_1 )
   END_RUNG
   RUNG wire#w1
      R_Coil( "MARCAS CIP".RUN_CIP_TANQUE_17 )
   END_RUNG
   RUNG wire#w1
      R_Coil( "MARCAS CIP".RUN_CIP_FONDO_TQ17 )
   END_RUNG
   RUNG wire#w1
      R_Coil( "MARCAS CIP".RUN_CIP_TANQUE_20 )
   END_RUNG
   RUNG wire#w1
      R_Coil( "MARCAS CIP".RUN_CIP_LINEA_TANQUE20 )
   END_RUNG
   RUNG wire#w1
      R_Coil( "MARCAS CIP".RUN_CIP_TQ20_MIXER2 )
   END_RUNG
   RUNG wire#w1
      R_Coil( "MARCAS CIP".RUN_CIP_LINEA_MIXER2 )
   END_RUNG
   RUNG wire#w1
      R_Coil( "MARCAS CIP".RUN_CIP_TANQUE_2 )
   END_RUNG
   RUNG wire#w1
      R_Coil( "MARCAS CIP".RUN_CIP_LINEA_TANQUE_1 )
   END_RUNG
   RUNG wire#w1
      R_Coil( "MARCAS CIP".RUN_CIP_LINEA_TANQUE_2 )
   END_RUNG
   RUNG wire#w1
      R_Coil( "MARCAS CIP".RUN_CIP_L_DESCARGA_LECHE )
   END_RUNG
   RUNG wire#w1
      R_Coil( "MARCAS CIP".RUN_CIP_TANQUE_3 )
   END_RUNG
   RUNG wire#w1
      R_Coil( "MARCAS CIP".RUN_CIP_TANQUE_4 )
   END_RUNG
   RUNG wire#w1
      R_Coil( "MARCAS CIP".RUN_CIP_MEZ_NATILLAS )
   END_RUNG
   RUNG wire#w1
      R_Coil( "MARCAS CIP".RUN_CIP_L_LECHE_MEZCLAS )
   END_RUNG
   RUNG wire#w1
      R_Coil( "MARCAS CIP".RUN_CIP_TANQUE_12 )
   END_RUNG
   RUNG wire#w1
      R_Coil( "MARCAS CIP".RUN_CIP_AMASADORA_1 )
   END_RUNG
   RUNG wire#w1
      R_Coil( "MARCAS CIP".RUN_CIP_BATIDOR_1 )
   END_RUNG
   RUNG wire#w1
      R_Coil( "MARCAS CIP".RUN_CIP_BATIDOR_Y_CLARA )
   END_RUNG
   RUNG wire#w1
      R_Coil( "MARCAS CIP".RUN_CIP_TANQUE_13 )
   END_RUNG
   RUNG wire#w1
      R_Coil( "MARCAS CIP".RUN_CIP_AMASADORA_2 )
   END_RUNG
   RUNG wire#w1
      R_Coil( "MARCAS CIP".RUN_CIP_BATIDOR_Y_CLARA2 )
   END_RUNG
   RUNG wire#w1
      R_Coil( "MARCAS CIP".RUN_CIP_PASTE )
   END_RUNG
   RUNG wire#w1
      R_Coil( "MARCAS CIP".RUN_CIP_L_LECHE_A_FLAN )
   END_RUNG
   RUNG wire#w1
      R_Coil( "MARCAS CIP".RUN_CIP_L_LECHE_NATILLAS )
   END_RUNG
   RUNG wire#w1
      R_Coil( "MARCAS CIP".RUN_CIP_L_PASTE_A_TQ9 )
   END_RUNG
   RUNG wire#w1
      R_Coil( "MARCAS CIP".RUN_CIP_L_PREPASTE )
   END_RUNG
   RUNG wire#w1
      R_Coil( "MARCAS CIP".MARCHA_CIP_LINEA_1 )
   END_RUNG
   RUNG wire#w1
      R_Coil( "MARCAS CIP".RUN_CIP_TQ_21_S_LACTOSA )
   END_RUNG
   RUNG wire#w1
      R_Coil( "M_RUN_CIP_TQ21" )
   END_RUNG
   // the same network as SCL:
   #_w1 := "PASOS CIP L1".paso_02_vaciado_tanque AND "MARCAS CIP".SELECCION_CIP_AGUA_L1 AND "Tag_752" AND NOT "DETECTOR FLUJO RET_L1";
   IF #_w1 THEN
       "PASOS CIP L1".paso_02_vaciado_tanque := FALSE;
       "MARCAS CIP".RUN_CIP_TANQUE_1 := FALSE;
       "MARCAS CIP".RUN_CIP_TANQUE_17 := FALSE;
       "MARCAS CIP".RUN_CIP_FONDO_TQ17 := FALSE;
       "MARCAS CIP".RUN_CIP_TANQUE_20 := FALSE;
       "MARCAS CIP".RUN_CIP_LINEA_TANQUE20 := FALSE;
       "MARCAS CIP".RUN_CIP_TQ20_MIXER2 := FALSE;
       "MARCAS CIP".RUN_CIP_LINEA_MIXER2 := FALSE;
       "MARCAS CIP".RUN_CIP_TANQUE_2 := FALSE;
       "MARCAS CIP".RUN_CIP_LINEA_TANQUE_1 := FALSE;
       "MARCAS CIP".RUN_CIP_LINEA_TANQUE_2 := FALSE;
       "MARCAS CIP".RUN_CIP_L_DESCARGA_LECHE := FALSE;
       "MARCAS CIP".RUN_CIP_TANQUE_3 := FALSE;
       "MARCAS CIP".RUN_CIP_TANQUE_4 := FALSE;
       "MARCAS CIP".RUN_CIP_MEZ_NATILLAS := FALSE;
       "MARCAS CIP".RUN_CIP_L_LECHE_MEZCLAS := FALSE;
       "MARCAS CIP".RUN_CIP_TANQUE_12 := FALSE;
       "MARCAS CIP".RUN_CIP_AMASADORA_1 := FALSE;
       "MARCAS CIP".RUN_CIP_BATIDOR_1 := FALSE;
       "MARCAS CIP".RUN_CIP_BATIDOR_Y_CLARA := FALSE;
       "MARCAS CIP".RUN_CIP_TANQUE_13 := FALSE;
       "MARCAS CIP".RUN_CIP_AMASADORA_2 := FALSE;
       "MARCAS CIP".RUN_CIP_BATIDOR_Y_CLARA2 := FALSE;
       "MARCAS CIP".RUN_CIP_PASTE := FALSE;
       "MARCAS CIP".RUN_CIP_L_LECHE_A_FLAN := FALSE;
       "MARCAS CIP".RUN_CIP_L_LECHE_NATILLAS := FALSE;
       "MARCAS CIP".RUN_CIP_L_PASTE_A_TQ9 := FALSE;
       "MARCAS CIP".RUN_CIP_L_PREPASTE := FALSE;
       "MARCAS CIP".MARCHA_CIP_LINEA_1 := FALSE;
       "MARCAS CIP".RUN_CIP_TQ_21_S_LACTOSA := FALSE;
       "M_RUN_CIP_TQ21" := FALSE;
   END_IF;
END_REGION

REGION Network 16
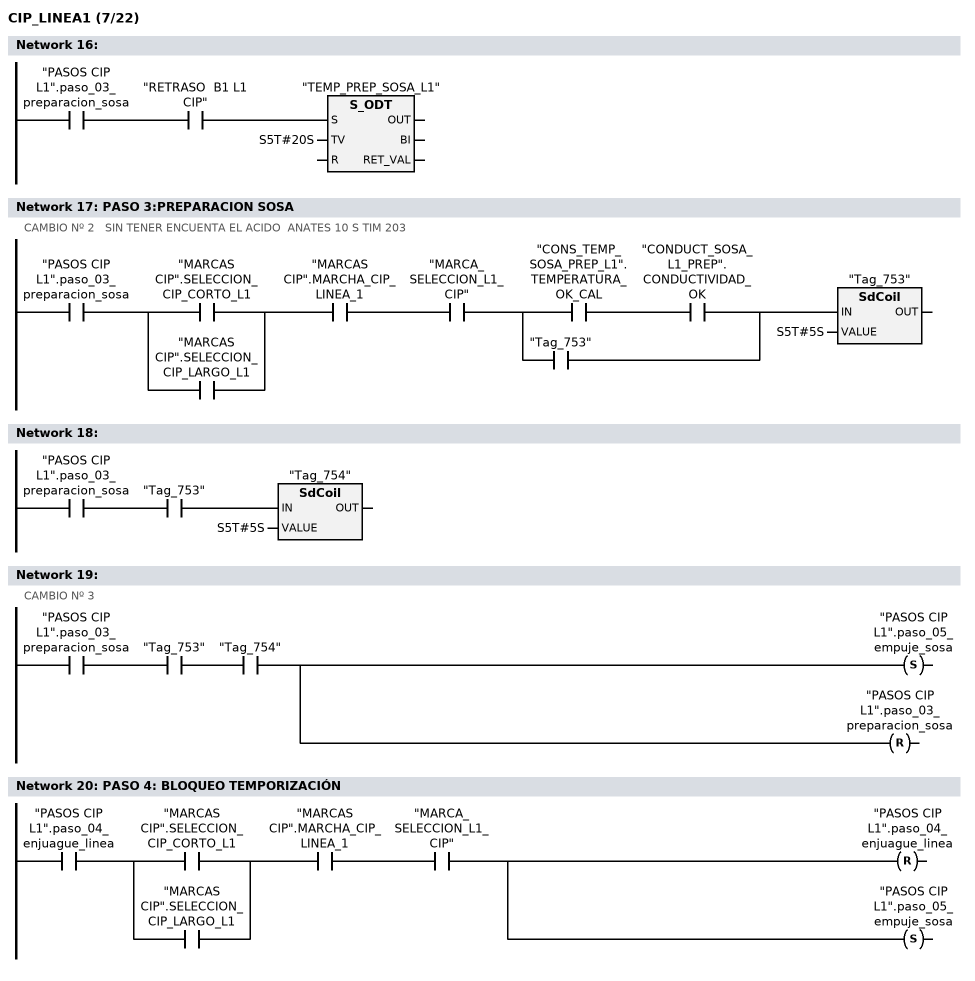
   RUNG wire#powerrail
      Contact( "PASOS CIP L1".paso_03_preparacion_sosa )
      Contact( "RETRASO  B1 L1 CIP" )
      S_ODT(T_NO := "TEMP_PREP_SOSA_L1", TV := S5T#20S, R :=, BI =>, RET_VAL =>)
   END_RUNG
   // the same network as SCL:
   #_s5time1 := S_ODT(T_NO := "TEMP_PREP_SOSA_L1",
                      TV := S5T#20S,
                      S := "PASOS CIP L1".paso_03_preparacion_sosa AND "RETRASO  B1 L1 CIP");
END_REGION

REGION Network 17: PASO 3:PREPARACION SOSA
   // CAMBIO Nº 2   SIN TENER ENCUENTA EL ACIDO  ANATES 10 S TIM 203
   // no SCL statement known for SdCoil: written as a call
   SdCoil(value := S5T#5S,
          in := "PASOS CIP L1".paso_03_preparacion_sosa AND ("MARCAS CIP".SELECCION_CIP_CORTO_L1 OR "MARCAS CIP".SELECCION_CIP_LARGO_L1) AND "MARCAS CIP".MARCHA_CIP_LINEA_1 AND "MARCA_SELECCION_L1_CIP" AND (("CONS_TEMP_SOSA_PREP_L1".TEMPERATURA_OK_CAL AND "CONDUCT_SOSA_L1_PREP".CONDUCTIVIDAD_OK) OR "Tag_753"),
          operand := "Tag_753");
END_REGION

REGION Network 18
   // no SCL statement known for SdCoil: written as a call
   SdCoil(value := S5T#5S, operand := "Tag_754", in := "PASOS CIP L1".paso_03_preparacion_sosa AND "Tag_753");
END_REGION

REGION Network 19
   // CAMBIO Nº 3
   RUNG wire#powerrail
      Contact( "PASOS CIP L1".paso_03_preparacion_sosa )
      Contact( "Tag_753" )
      Contact( "Tag_754" )
      wire#w1
      S_Coil( "PASOS CIP L1".paso_05_empuje_sosa )
   END_RUNG
   RUNG wire#w1
      R_Coil( "PASOS CIP L1".paso_03_preparacion_sosa )
   END_RUNG
   // the same network as SCL:
   IF "PASOS CIP L1".paso_03_preparacion_sosa AND "Tag_753" AND "Tag_754" THEN
       "PASOS CIP L1".paso_05_empuje_sosa := TRUE;
       "PASOS CIP L1".paso_03_preparacion_sosa := FALSE;
   END_IF;
END_REGION

REGION Network 20: PASO 4: BLOQUEO TEMPORIZACIÓN
   RUNG wire#powerrail
      Contact( "PASOS CIP L1".paso_04_enjuague_linea )
      wire#w1
      Contact( "MARCAS CIP".SELECCION_CIP_CORTO_L1 )
      wire#w2
      Contact( "MARCAS CIP".MARCHA_CIP_LINEA_1 )
      Contact( "MARCA_SELECCION_L1_CIP" )
      wire#w3
      R_Coil( "PASOS CIP L1".paso_04_enjuague_linea )
   END_RUNG
   RUNG wire#w1
      Contact( "MARCAS CIP".SELECCION_CIP_LARGO_L1 )
   END_RUNG wire#w2
   RUNG wire#w3
      S_Coil( "PASOS CIP L1".paso_05_empuje_sosa )
   END_RUNG
   // the same network as SCL:
   #_w1 := "PASOS CIP L1".paso_04_enjuague_linea AND ("MARCAS CIP".SELECCION_CIP_CORTO_L1 OR "MARCAS CIP".SELECCION_CIP_LARGO_L1) AND "MARCAS CIP".MARCHA_CIP_LINEA_1 AND "MARCA_SELECCION_L1_CIP";
   IF #_w1 THEN
       "PASOS CIP L1".paso_04_enjuague_linea := FALSE;
       "PASOS CIP L1".paso_05_empuje_sosa := TRUE;
   END_IF;
END_REGION

REGION Network 21: PASO 5: EMPUJE SOSA
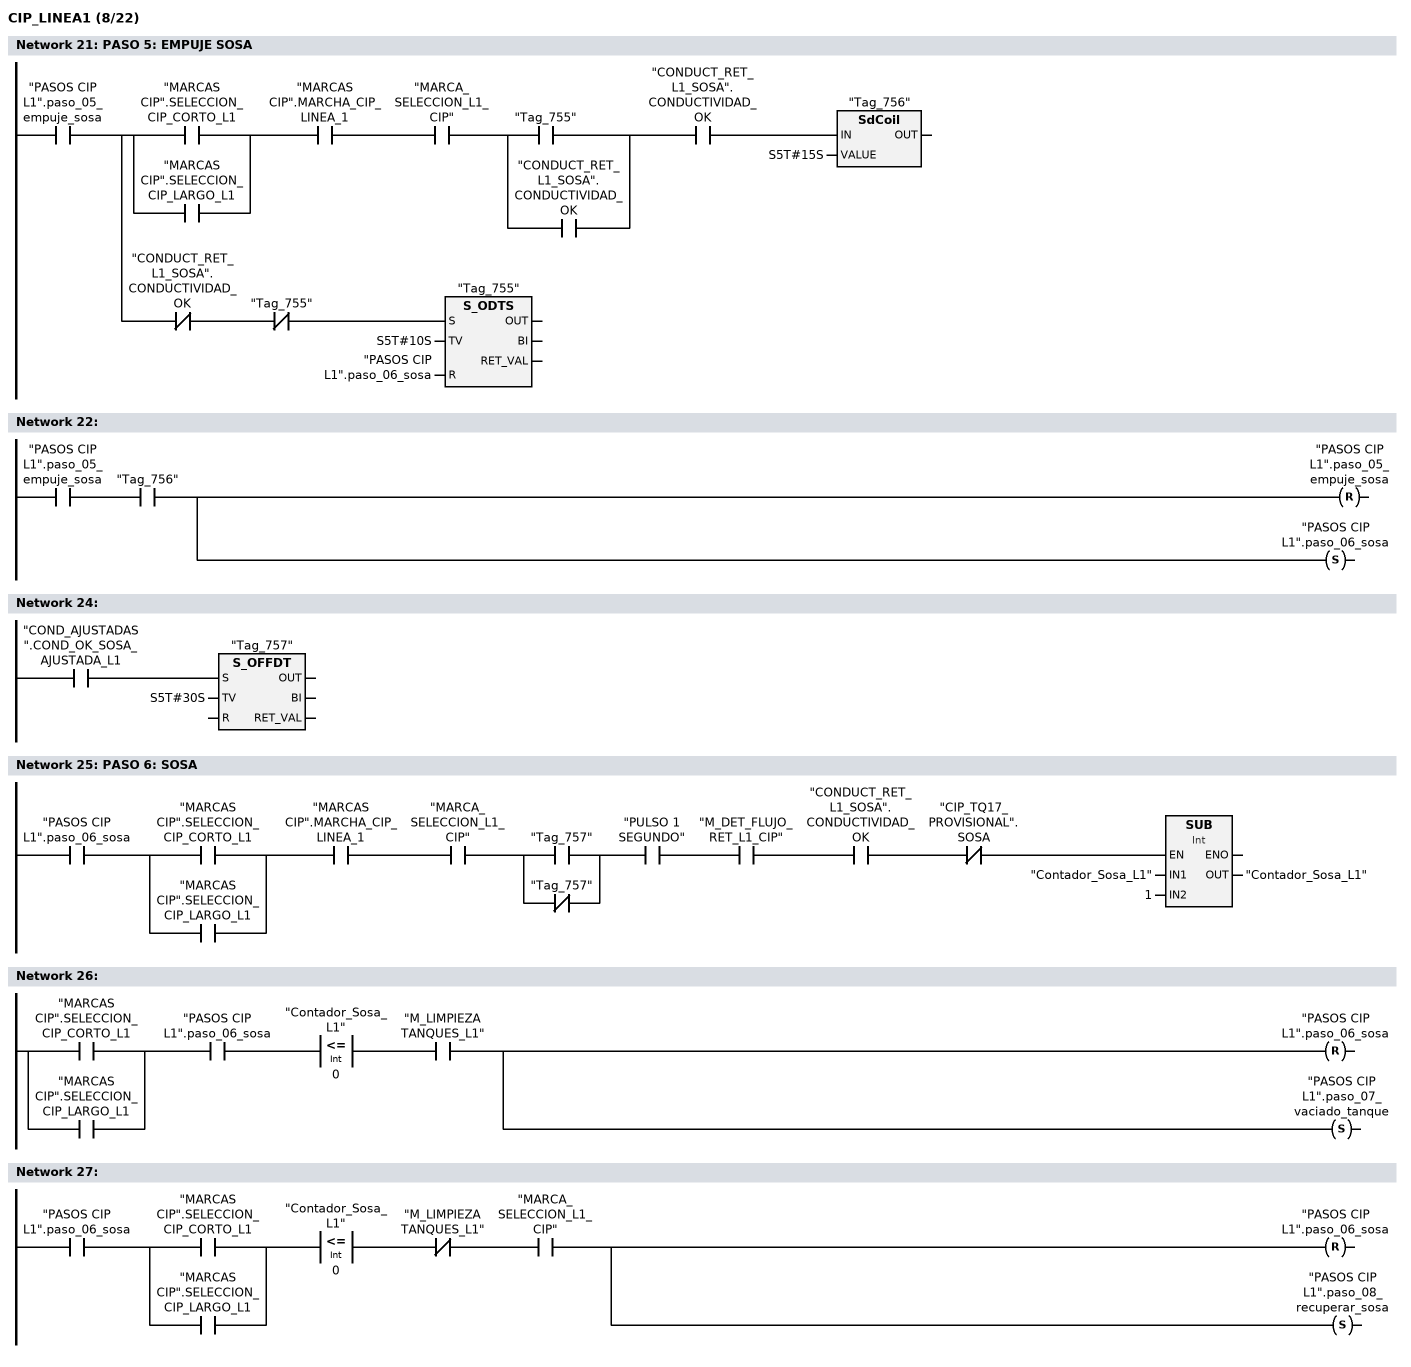
   // no SCL statement known for SdCoil: written as a call
   #_w1 := "PASOS CIP L1".paso_05_empuje_sosa;
   SdCoil(value := S5T#15S,
          operand := "Tag_756",
          in := "PASOS CIP L1".paso_05_empuje_sosa AND ("MARCAS CIP".SELECCION_CIP_CORTO_L1 OR "MARCAS CIP".SELECCION_CIP_LARGO_L1) AND "MARCAS CIP".MARCHA_CIP_LINEA_1 AND "MARCA_SELECCION_L1_CIP" AND ("Tag_755" OR "CONDUCT_RET_L1_SOSA".CONDUCTIVIDAD_OK) AND "CONDUCT_RET_L1_SOSA".CONDUCTIVIDAD_OK);
   #_s5time1 := S_ODTS(T_NO := "Tag_755",
                       TV := S5T#10S,
                       R := "PASOS CIP L1".paso_06_sosa,
                       S := #_w1 AND NOT "CONDUCT_RET_L1_SOSA".CONDUCTIVIDAD_OK AND NOT "Tag_755");
END_REGION

REGION Network 22
   RUNG wire#powerrail
      Contact( "PASOS CIP L1".paso_05_empuje_sosa )
      Contact( "Tag_756" )
      wire#w1
      R_Coil( "PASOS CIP L1".paso_05_empuje_sosa )
   END_RUNG
   RUNG wire#w1
      S_Coil( "PASOS CIP L1".paso_06_sosa )
   END_RUNG
   // the same network as SCL:
   #_w1 := "PASOS CIP L1".paso_05_empuje_sosa AND "Tag_756";
   IF #_w1 THEN
       "PASOS CIP L1".paso_05_empuje_sosa := FALSE;
       "PASOS CIP L1".paso_06_sosa := TRUE;
   END_IF;
END_REGION

NETWORK
TITLE = 
      A     "PASOS CIP L1".paso_06_sosa;
      JC    c1;
      L     "SP TIM L1 CIP".TIM_PASO_6_L1;
      L     60;
      *I;
      T     "Contador_Sosa_L1";
c1:   NOP   0;

REGION Network 24
   RUNG wire#powerrail
      Contact( "COND_AJUSTADAS".COND_OK_SOSA_AJUSTADA_L1 )
      S_OFFDT(T_NO := "Tag_757", TV := S5T#30S, R :=, BI =>, RET_VAL =>)
   END_RUNG
   // the same network as SCL:
   #_s5time1 := S_OFFDT(T_NO := "Tag_757", TV := S5T#30S, S := "COND_AJUSTADAS".COND_OK_SOSA_AJUSTADA_L1);
END_REGION

REGION Network 25: PASO 6: SOSA
   RUNG wire#powerrail
      Contact( "PASOS CIP L1".paso_06_sosa )
      wire#w1
      Contact( "MARCAS CIP".SELECCION_CIP_CORTO_L1 )
      wire#w2
      Contact( "MARCAS CIP".MARCHA_CIP_LINEA_1 )
      Contact( "MARCA_SELECCION_L1_CIP" )
      wire#w3
      Contact( "Tag_757" )
      wire#w4
      Contact( "PULSO 1 SEGUNDO" )
      Contact( "M_DET_FLUJO_RET_L1_CIP" )
      Contact( "CONDUCT_RET_L1_SOSA".CONDUCTIVIDAD_OK )
      I_Contact( "CIP_TQ17_PROVISIONAL".SOSA )
      { S7_Templates := "SrcType := Int"; S7_GenerateENO := "TRUE" } Sub(in1 := "Contador_Sosa_L1", in2 := 1, out => "Contador_Sosa_L1")
   END_RUNG
   RUNG wire#w1
      Contact( "MARCAS CIP".SELECCION_CIP_LARGO_L1 )
   END_RUNG wire#w2
   RUNG wire#w3
      I_Contact( "Tag_757" )
   END_RUNG wire#w4
   // the same network as SCL:
   IF "PASOS CIP L1".paso_06_sosa AND ("MARCAS CIP".SELECCION_CIP_CORTO_L1 OR "MARCAS CIP".SELECCION_CIP_LARGO_L1) AND "MARCAS CIP".MARCHA_CIP_LINEA_1 AND "MARCA_SELECCION_L1_CIP" AND ("Tag_757" OR NOT "Tag_757") AND "PULSO 1 SEGUNDO" AND "M_DET_FLUJO_RET_L1_CIP" AND "CONDUCT_RET_L1_SOSA".CONDUCTIVIDAD_OK AND NOT "CIP_TQ17_PROVISIONAL".SOSA THEN
       "Contador_Sosa_L1" := "Contador_Sosa_L1" - 1;
   END_IF;
END_REGION

REGION Network 26
   RUNG wire#powerrail
      Contact( "MARCAS CIP".SELECCION_CIP_CORTO_L1 )
      wire#w1
      Contact( "PASOS CIP L1".paso_06_sosa )
      { S7_Templates := "SrcType := Int" } LE_Contact(in1 := "Contador_Sosa_L1", in2 := 0)
      Contact( "M_LIMPIEZA TANQUES_L1" )
      wire#w2
      R_Coil( "PASOS CIP L1".paso_06_sosa )
   END_RUNG
   RUNG wire#powerrail
      Contact( "MARCAS CIP".SELECCION_CIP_LARGO_L1 )
   END_RUNG wire#w1
   RUNG wire#w2
      S_Coil( "PASOS CIP L1".paso_07_vaciado_tanque )
   END_RUNG
   // the same network as SCL:
   #_w1 := ("MARCAS CIP".SELECCION_CIP_CORTO_L1 OR "MARCAS CIP".SELECCION_CIP_LARGO_L1) AND "PASOS CIP L1".paso_06_sosa AND ("Contador_Sosa_L1" <= 0) AND "M_LIMPIEZA TANQUES_L1";
   IF #_w1 THEN
       "PASOS CIP L1".paso_06_sosa := FALSE;
       "PASOS CIP L1".paso_07_vaciado_tanque := TRUE;
   END_IF;
END_REGION

REGION Network 27
   RUNG wire#powerrail
      Contact( "PASOS CIP L1".paso_06_sosa )
      wire#w1
      Contact( "MARCAS CIP".SELECCION_CIP_CORTO_L1 )
      wire#w2
      { S7_Templates := "SrcType := Int" } LE_Contact(in1 := "Contador_Sosa_L1", in2 := 0)
      I_Contact( "M_LIMPIEZA TANQUES_L1" )
      Contact( "MARCA_SELECCION_L1_CIP" )
      wire#w3
      R_Coil( "PASOS CIP L1".paso_06_sosa )
   END_RUNG
   RUNG wire#w1
      Contact( "MARCAS CIP".SELECCION_CIP_LARGO_L1 )
   END_RUNG wire#w2
   RUNG wire#w3
      S_Coil( "PASOS CIP L1".paso_08_recuperar_sosa )
   END_RUNG
   // the same network as SCL:
   #_w1 := "PASOS CIP L1".paso_06_sosa AND ("MARCAS CIP".SELECCION_CIP_CORTO_L1 OR "MARCAS CIP".SELECCION_CIP_LARGO_L1) AND ("Contador_Sosa_L1" <= 0) AND NOT "M_LIMPIEZA TANQUES_L1" AND "MARCA_SELECCION_L1_CIP";
   IF #_w1 THEN
       "PASOS CIP L1".paso_06_sosa := FALSE;
       "PASOS CIP L1".paso_08_recuperar_sosa := TRUE;
   END_IF;
END_REGION

REGION Network 28: PASO 7: VACIADO SI TANQUE
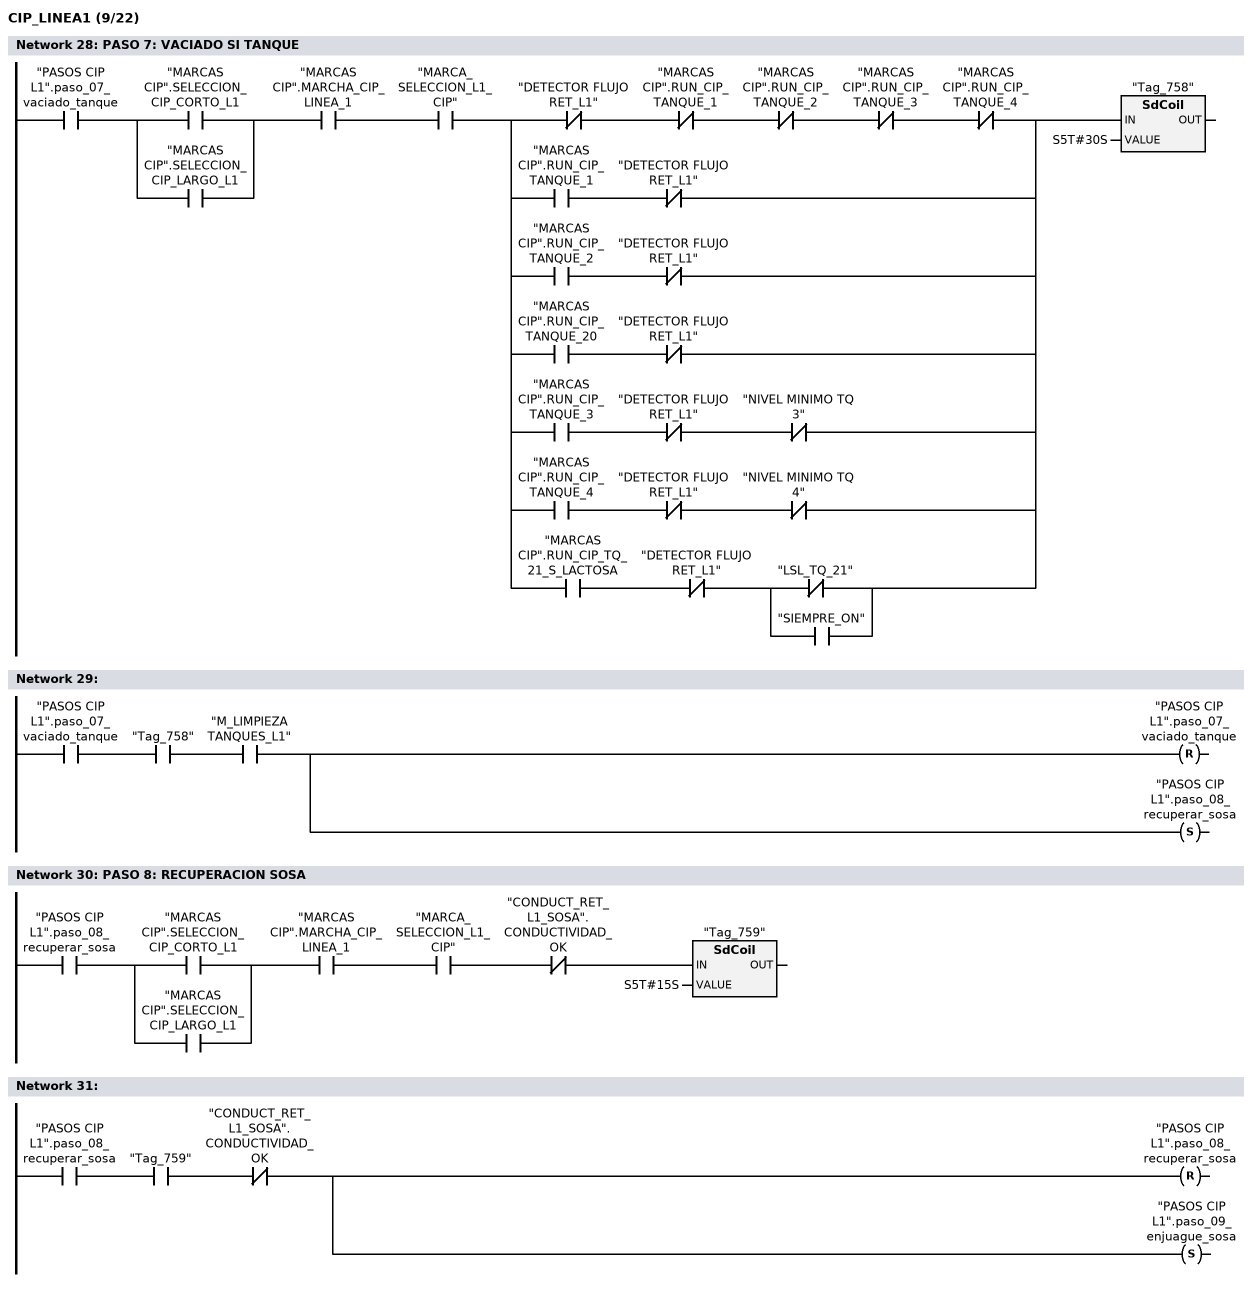
   // no SCL statement known for SdCoil: written as a call
   SdCoil(value := S5T#30S,
          in := "PASOS CIP L1".paso_07_vaciado_tanque AND ("MARCAS CIP".SELECCION_CIP_CORTO_L1 OR "MARCAS CIP".SELECCION_CIP_LARGO_L1) AND "MARCAS CIP".MARCHA_CIP_LINEA_1 AND "MARCA_SELECCION_L1_CIP" AND ((NOT "DETECTOR FLUJO RET_L1" AND NOT "MARCAS CIP".RUN_CIP_TANQUE_1 AND NOT "MARCAS CIP".RUN_CIP_TANQUE_2 AND NOT "MARCAS CIP".RUN_CIP_TANQUE_3 AND NOT "MARCAS CIP".RUN_CIP_TANQUE_4) OR ("MARCAS CIP".RUN_CIP_TANQUE_1 AND NOT "DETECTOR FLUJO RET_L1") OR ("MARCAS CIP".RUN_CIP_TANQUE_2 AND NOT "DETECTOR FLUJO RET_L1") OR ("MARCAS CIP".RUN_CIP_TANQUE_20 AND NOT "DETECTOR FLUJO RET_L1") OR ("MARCAS CIP".RUN_CIP_TANQUE_3 AND NOT "DETECTOR FLUJO RET_L1" AND NOT "NIVEL MINIMO TQ 3") OR ("MARCAS CIP".RUN_CIP_TANQUE_4 AND NOT "DETECTOR FLUJO RET_L1" AND NOT "NIVEL MINIMO TQ 4") OR ("MARCAS CIP".RUN_CIP_TQ_21_S_LACTOSA AND NOT "DETECTOR FLUJO RET_L1" AND (NOT "LSL_TQ_21" OR "SIEMPRE_ON"))),
          operand := "Tag_758");
END_REGION

REGION Network 29
   RUNG wire#powerrail
      Contact( "PASOS CIP L1".paso_07_vaciado_tanque )
      Contact( "Tag_758" )
      Contact( "M_LIMPIEZA TANQUES_L1" )
      wire#w1
      R_Coil( "PASOS CIP L1".paso_07_vaciado_tanque )
   END_RUNG
   RUNG wire#w1
      S_Coil( "PASOS CIP L1".paso_08_recuperar_sosa )
   END_RUNG
   // the same network as SCL:
   #_w1 := "PASOS CIP L1".paso_07_vaciado_tanque AND "Tag_758" AND "M_LIMPIEZA TANQUES_L1";
   IF #_w1 THEN
       "PASOS CIP L1".paso_07_vaciado_tanque := FALSE;
       "PASOS CIP L1".paso_08_recuperar_sosa := TRUE;
   END_IF;
END_REGION

REGION Network 30: PASO 8: RECUPERACION SOSA
   // no SCL statement known for SdCoil: written as a call
   SdCoil(value := S5T#15S,
          operand := "Tag_759",
          in := "PASOS CIP L1".paso_08_recuperar_sosa AND ("MARCAS CIP".SELECCION_CIP_CORTO_L1 OR "MARCAS CIP".SELECCION_CIP_LARGO_L1) AND "MARCAS CIP".MARCHA_CIP_LINEA_1 AND "MARCA_SELECCION_L1_CIP" AND NOT "CONDUCT_RET_L1_SOSA".CONDUCTIVIDAD_OK);
END_REGION

REGION Network 31
   RUNG wire#powerrail
      Contact( "PASOS CIP L1".paso_08_recuperar_sosa )
      Contact( "Tag_759" )
      I_Contact( "CONDUCT_RET_L1_SOSA".CONDUCTIVIDAD_OK )
      wire#w1
      R_Coil( "PASOS CIP L1".paso_08_recuperar_sosa )
   END_RUNG
   RUNG wire#w1
      S_Coil( "PASOS CIP L1".paso_09_enjuague_sosa )
   END_RUNG
   // the same network as SCL:
   #_w1 := "PASOS CIP L1".paso_08_recuperar_sosa AND "Tag_759" AND NOT "CONDUCT_RET_L1_SOSA".CONDUCTIVIDAD_OK;
   IF #_w1 THEN
       "PASOS CIP L1".paso_08_recuperar_sosa := FALSE;
       "PASOS CIP L1".paso_09_enjuague_sosa := TRUE;
   END_IF;
END_REGION

REGION Network 32: PASO 9: ENJUAGUE SOSA
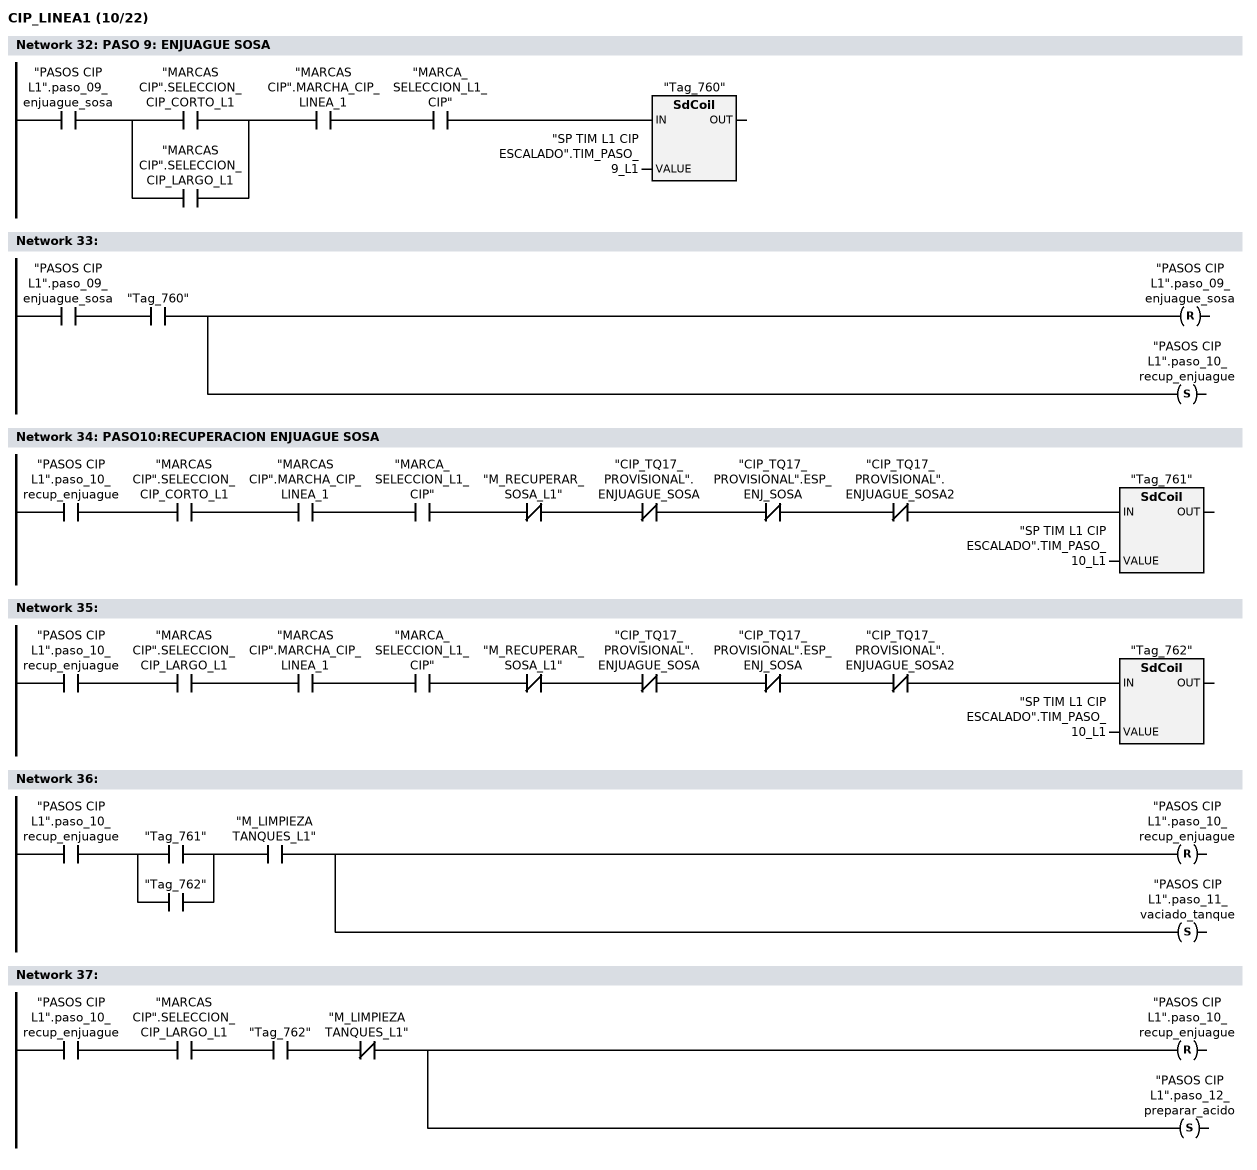
   // no SCL statement known for SdCoil: written as a call
   SdCoil(value := "SP TIM L1 CIP ESCALADO".TIM_PASO_9_L1,
          operand := "Tag_760",
          in := "PASOS CIP L1".paso_09_enjuague_sosa AND ("MARCAS CIP".SELECCION_CIP_CORTO_L1 OR "MARCAS CIP".SELECCION_CIP_LARGO_L1) AND "MARCAS CIP".MARCHA_CIP_LINEA_1 AND "MARCA_SELECCION_L1_CIP");
END_REGION

REGION Network 33
   RUNG wire#powerrail
      Contact( "PASOS CIP L1".paso_09_enjuague_sosa )
      Contact( "Tag_760" )
      wire#w1
      R_Coil( "PASOS CIP L1".paso_09_enjuague_sosa )
   END_RUNG
   RUNG wire#w1
      S_Coil( "PASOS CIP L1".paso_10_recup_enjuague )
   END_RUNG
   // the same network as SCL:
   #_w1 := "PASOS CIP L1".paso_09_enjuague_sosa AND "Tag_760";
   IF #_w1 THEN
       "PASOS CIP L1".paso_09_enjuague_sosa := FALSE;
       "PASOS CIP L1".paso_10_recup_enjuague := TRUE;
   END_IF;
END_REGION

REGION Network 34: PASO10:RECUPERACION ENJUAGUE SOSA
   // no SCL statement known for SdCoil: written as a call
   SdCoil(value := "SP TIM L1 CIP ESCALADO".TIM_PASO_10_L1,
          operand := "Tag_761",
          in := "PASOS CIP L1".paso_10_recup_enjuague AND "MARCAS CIP".SELECCION_CIP_CORTO_L1 AND "MARCAS CIP".MARCHA_CIP_LINEA_1 AND "MARCA_SELECCION_L1_CIP" AND NOT "M_RECUPERAR_SOSA_L1" AND NOT "CIP_TQ17_PROVISIONAL".ENJUAGUE_SOSA AND NOT "CIP_TQ17_PROVISIONAL".ESP_ENJ_SOSA AND NOT "CIP_TQ17_PROVISIONAL".ENJUAGUE_SOSA2);
END_REGION

REGION Network 35
   // no SCL statement known for SdCoil: written as a call
   SdCoil(value := "SP TIM L1 CIP ESCALADO".TIM_PASO_10_L1,
          operand := "Tag_762",
          in := "PASOS CIP L1".paso_10_recup_enjuague AND "MARCAS CIP".SELECCION_CIP_LARGO_L1 AND "MARCAS CIP".MARCHA_CIP_LINEA_1 AND "MARCA_SELECCION_L1_CIP" AND NOT "M_RECUPERAR_SOSA_L1" AND NOT "CIP_TQ17_PROVISIONAL".ENJUAGUE_SOSA AND NOT "CIP_TQ17_PROVISIONAL".ESP_ENJ_SOSA AND NOT "CIP_TQ17_PROVISIONAL".ENJUAGUE_SOSA2);
END_REGION

REGION Network 36
   RUNG wire#powerrail
      Contact( "PASOS CIP L1".paso_10_recup_enjuague )
      wire#w1
      Contact( "Tag_761" )
      wire#w2
      Contact( "M_LIMPIEZA TANQUES_L1" )
      wire#w3
      R_Coil( "PASOS CIP L1".paso_10_recup_enjuague )
   END_RUNG
   RUNG wire#w1
      Contact( "Tag_762" )
   END_RUNG wire#w2
   RUNG wire#w3
      S_Coil( "PASOS CIP L1".paso_11_vaciado_tanque )
   END_RUNG
   // the same network as SCL:
   #_w1 := "PASOS CIP L1".paso_10_recup_enjuague AND ("Tag_761" OR "Tag_762") AND "M_LIMPIEZA TANQUES_L1";
   IF #_w1 THEN
       "PASOS CIP L1".paso_10_recup_enjuague := FALSE;
       "PASOS CIP L1".paso_11_vaciado_tanque := TRUE;
   END_IF;
END_REGION

REGION Network 37
   RUNG wire#powerrail
      Contact( "PASOS CIP L1".paso_10_recup_enjuague )
      Contact( "MARCAS CIP".SELECCION_CIP_LARGO_L1 )
      Contact( "Tag_762" )
      I_Contact( "M_LIMPIEZA TANQUES_L1" )
      wire#w1
      R_Coil( "PASOS CIP L1".paso_10_recup_enjuague )
   END_RUNG
   RUNG wire#w1
      S_Coil( "PASOS CIP L1".paso_12_preparar_acido )
   END_RUNG
   // the same network as SCL:
   #_w1 := "PASOS CIP L1".paso_10_recup_enjuague AND "MARCAS CIP".SELECCION_CIP_LARGO_L1 AND "Tag_762" AND NOT "M_LIMPIEZA TANQUES_L1";
   IF #_w1 THEN
       "PASOS CIP L1".paso_10_recup_enjuague := FALSE;
       "PASOS CIP L1".paso_12_preparar_acido := TRUE;
   END_IF;
END_REGION

REGION Network 38
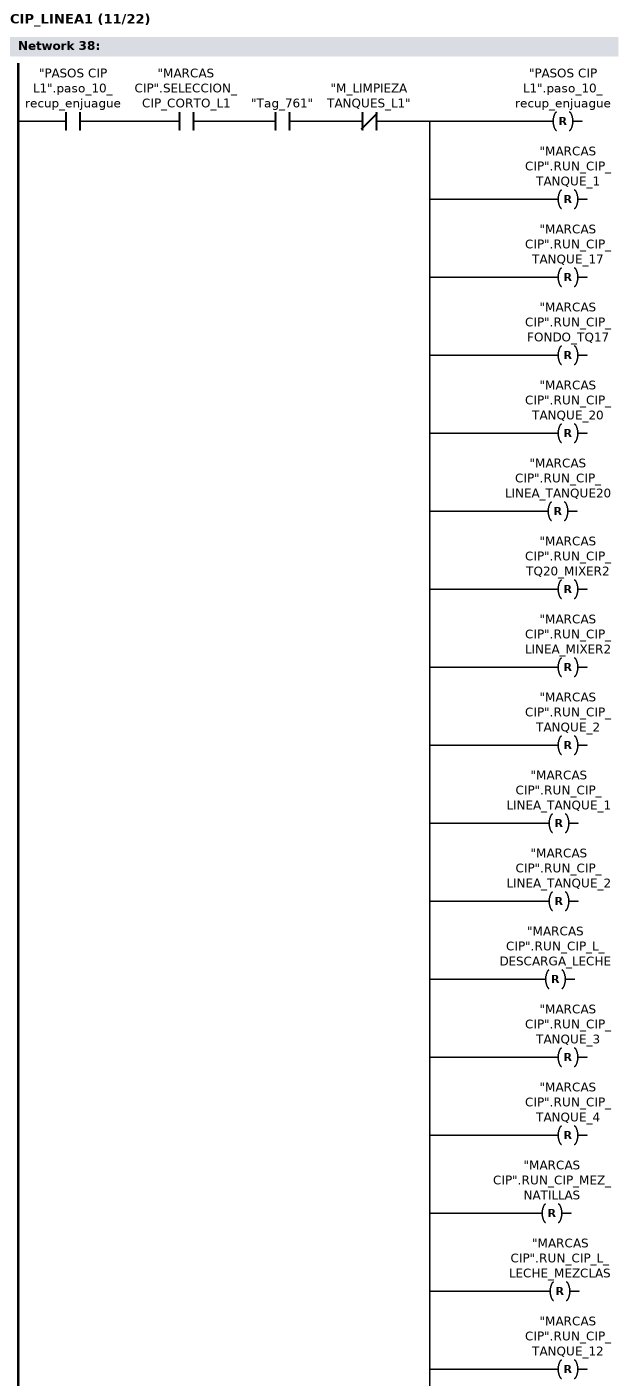
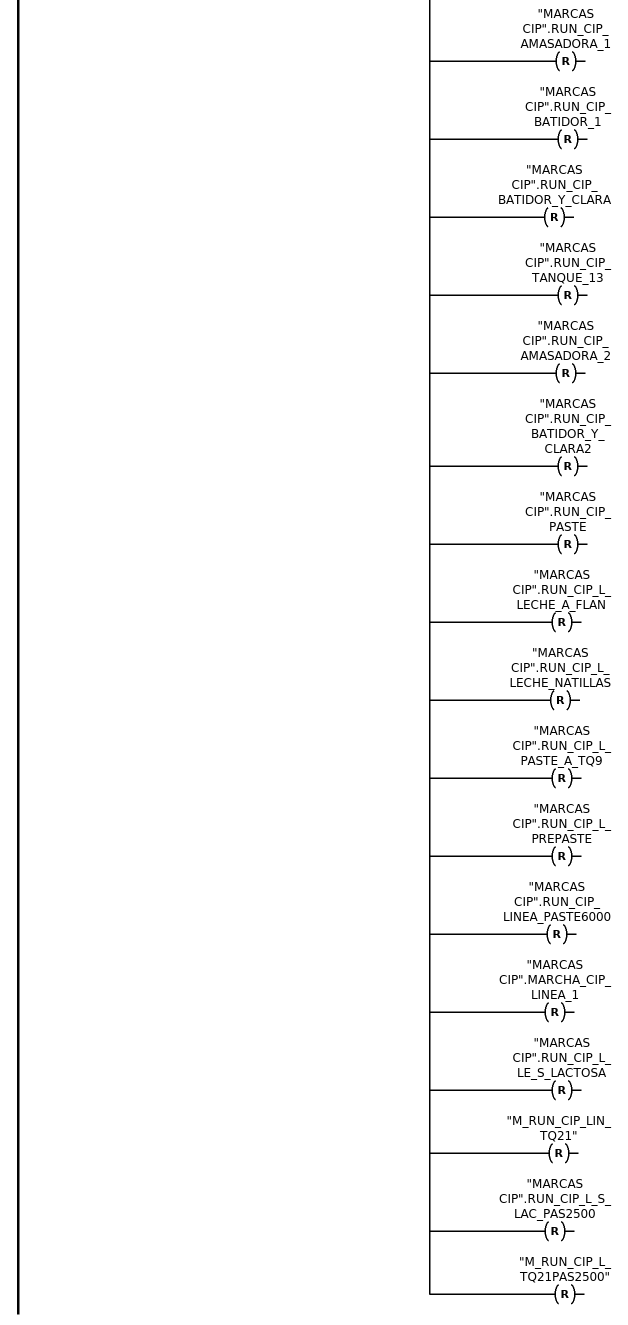
   RUNG wire#powerrail
      Contact( "PASOS CIP L1".paso_10_recup_enjuague )
      Contact( "MARCAS CIP".SELECCION_CIP_CORTO_L1 )
      Contact( "Tag_761" )
      I_Contact( "M_LIMPIEZA TANQUES_L1" )
      wire#w1
      R_Coil( "PASOS CIP L1".paso_10_recup_enjuague )
   END_RUNG
   RUNG wire#w1
      R_Coil( "MARCAS CIP".RUN_CIP_TANQUE_1 )
   END_RUNG
   RUNG wire#w1
      R_Coil( "MARCAS CIP".RUN_CIP_TANQUE_17 )
   END_RUNG
   RUNG wire#w1
      R_Coil( "MARCAS CIP".RUN_CIP_FONDO_TQ17 )
   END_RUNG
   RUNG wire#w1
      R_Coil( "MARCAS CIP".RUN_CIP_TANQUE_20 )
   END_RUNG
   RUNG wire#w1
      R_Coil( "MARCAS CIP".RUN_CIP_LINEA_TANQUE20 )
   END_RUNG
   RUNG wire#w1
      R_Coil( "MARCAS CIP".RUN_CIP_TQ20_MIXER2 )
   END_RUNG
   RUNG wire#w1
      R_Coil( "MARCAS CIP".RUN_CIP_LINEA_MIXER2 )
   END_RUNG
   RUNG wire#w1
      R_Coil( "MARCAS CIP".RUN_CIP_TANQUE_2 )
   END_RUNG
   RUNG wire#w1
      R_Coil( "MARCAS CIP".RUN_CIP_LINEA_TANQUE_1 )
   END_RUNG
   RUNG wire#w1
      R_Coil( "MARCAS CIP".RUN_CIP_LINEA_TANQUE_2 )
   END_RUNG
   RUNG wire#w1
      R_Coil( "MARCAS CIP".RUN_CIP_L_DESCARGA_LECHE )
   END_RUNG
   RUNG wire#w1
      R_Coil( "MARCAS CIP".RUN_CIP_TANQUE_3 )
   END_RUNG
   RUNG wire#w1
      R_Coil( "MARCAS CIP".RUN_CIP_TANQUE_4 )
   END_RUNG
   RUNG wire#w1
      R_Coil( "MARCAS CIP".RUN_CIP_MEZ_NATILLAS )
   END_RUNG
   RUNG wire#w1
      R_Coil( "MARCAS CIP".RUN_CIP_L_LECHE_MEZCLAS )
   END_RUNG
   RUNG wire#w1
      R_Coil( "MARCAS CIP".RUN_CIP_TANQUE_12 )
   END_RUNG
   RUNG wire#w1
      R_Coil( "MARCAS CIP".RUN_CIP_AMASADORA_1 )
   END_RUNG
   RUNG wire#w1
      R_Coil( "MARCAS CIP".RUN_CIP_BATIDOR_1 )
   END_RUNG
   RUNG wire#w1
      R_Coil( "MARCAS CIP".RUN_CIP_BATIDOR_Y_CLARA )
   END_RUNG
   RUNG wire#w1
      R_Coil( "MARCAS CIP".RUN_CIP_TANQUE_13 )
   END_RUNG
   RUNG wire#w1
      R_Coil( "MARCAS CIP".RUN_CIP_AMASADORA_2 )
   END_RUNG
   RUNG wire#w1
      R_Coil( "MARCAS CIP".RUN_CIP_BATIDOR_Y_CLARA2 )
   END_RUNG
   RUNG wire#w1
      R_Coil( "MARCAS CIP".RUN_CIP_PASTE )
   END_RUNG
   RUNG wire#w1
      R_Coil( "MARCAS CIP".RUN_CIP_L_LECHE_A_FLAN )
   END_RUNG
   RUNG wire#w1
      R_Coil( "MARCAS CIP".RUN_CIP_L_LECHE_NATILLAS )
   END_RUNG
   RUNG wire#w1
      R_Coil( "MARCAS CIP".RUN_CIP_L_PASTE_A_TQ9 )
   END_RUNG
   RUNG wire#w1
      R_Coil( "MARCAS CIP".RUN_CIP_L_PREPASTE )
   END_RUNG
   RUNG wire#w1
      R_Coil( "MARCAS CIP".RUN_CIP_LINEA_PASTE6000 )
   END_RUNG
   RUNG wire#w1
      R_Coil( "MARCAS CIP".MARCHA_CIP_LINEA_1 )
   END_RUNG
   RUNG wire#w1
      R_Coil( "MARCAS CIP".RUN_CIP_L_LE_S_LACTOSA )
   END_RUNG
   RUNG wire#w1
      R_Coil( "M_RUN_CIP_LIN_TQ21" )
   END_RUNG
   RUNG wire#w1
      R_Coil( "MARCAS CIP".RUN_CIP_L_S_LAC_PAS2500 )
   END_RUNG
   RUNG wire#w1
      R_Coil( "M_RUN_CIP_L_TQ21PAS2500" )
   END_RUNG
   // the same network as SCL:
   #_w1 := "PASOS CIP L1".paso_10_recup_enjuague AND "MARCAS CIP".SELECCION_CIP_CORTO_L1 AND "Tag_761" AND NOT "M_LIMPIEZA TANQUES_L1";
   IF #_w1 THEN
       "PASOS CIP L1".paso_10_recup_enjuague := FALSE;
       "MARCAS CIP".RUN_CIP_TANQUE_1 := FALSE;
       "MARCAS CIP".RUN_CIP_TANQUE_17 := FALSE;
       "MARCAS CIP".RUN_CIP_FONDO_TQ17 := FALSE;
       "MARCAS CIP".RUN_CIP_TANQUE_20 := FALSE;
       "MARCAS CIP".RUN_CIP_LINEA_TANQUE20 := FALSE;
       "MARCAS CIP".RUN_CIP_TQ20_MIXER2 := FALSE;
       "MARCAS CIP".RUN_CIP_LINEA_MIXER2 := FALSE;
       "MARCAS CIP".RUN_CIP_TANQUE_2 := FALSE;
       "MARCAS CIP".RUN_CIP_LINEA_TANQUE_1 := FALSE;
       "MARCAS CIP".RUN_CIP_LINEA_TANQUE_2 := FALSE;
       "MARCAS CIP".RUN_CIP_L_DESCARGA_LECHE := FALSE;
       "MARCAS CIP".RUN_CIP_TANQUE_3 := FALSE;
       "MARCAS CIP".RUN_CIP_TANQUE_4 := FALSE;
       "MARCAS CIP".RUN_CIP_MEZ_NATILLAS := FALSE;
       "MARCAS CIP".RUN_CIP_L_LECHE_MEZCLAS := FALSE;
       "MARCAS CIP".RUN_CIP_TANQUE_12 := FALSE;
       "MARCAS CIP".RUN_CIP_AMASADORA_1 := FALSE;
       "MARCAS CIP".RUN_CIP_BATIDOR_1 := FALSE;
       "MARCAS CIP".RUN_CIP_BATIDOR_Y_CLARA := FALSE;
       "MARCAS CIP".RUN_CIP_TANQUE_13 := FALSE;
       "MARCAS CIP".RUN_CIP_AMASADORA_2 := FALSE;
       "MARCAS CIP".RUN_CIP_BATIDOR_Y_CLARA2 := FALSE;
       "MARCAS CIP".RUN_CIP_PASTE := FALSE;
       "MARCAS CIP".RUN_CIP_L_LECHE_A_FLAN := FALSE;
       "MARCAS CIP".RUN_CIP_L_LECHE_NATILLAS := FALSE;
       "MARCAS CIP".RUN_CIP_L_PASTE_A_TQ9 := FALSE;
       "MARCAS CIP".RUN_CIP_L_PREPASTE := FALSE;
       "MARCAS CIP".RUN_CIP_LINEA_PASTE6000 := FALSE;
       "MARCAS CIP".MARCHA_CIP_LINEA_1 := FALSE;
       "MARCAS CIP".RUN_CIP_L_LE_S_LACTOSA := FALSE;
       "M_RUN_CIP_LIN_TQ21" := FALSE;
       "MARCAS CIP".RUN_CIP_L_S_LAC_PAS2500 := FALSE;
       "M_RUN_CIP_L_TQ21PAS2500" := FALSE;
   END_IF;
END_REGION

REGION Network 39: PASO 11: VACIADO SI TANQUE
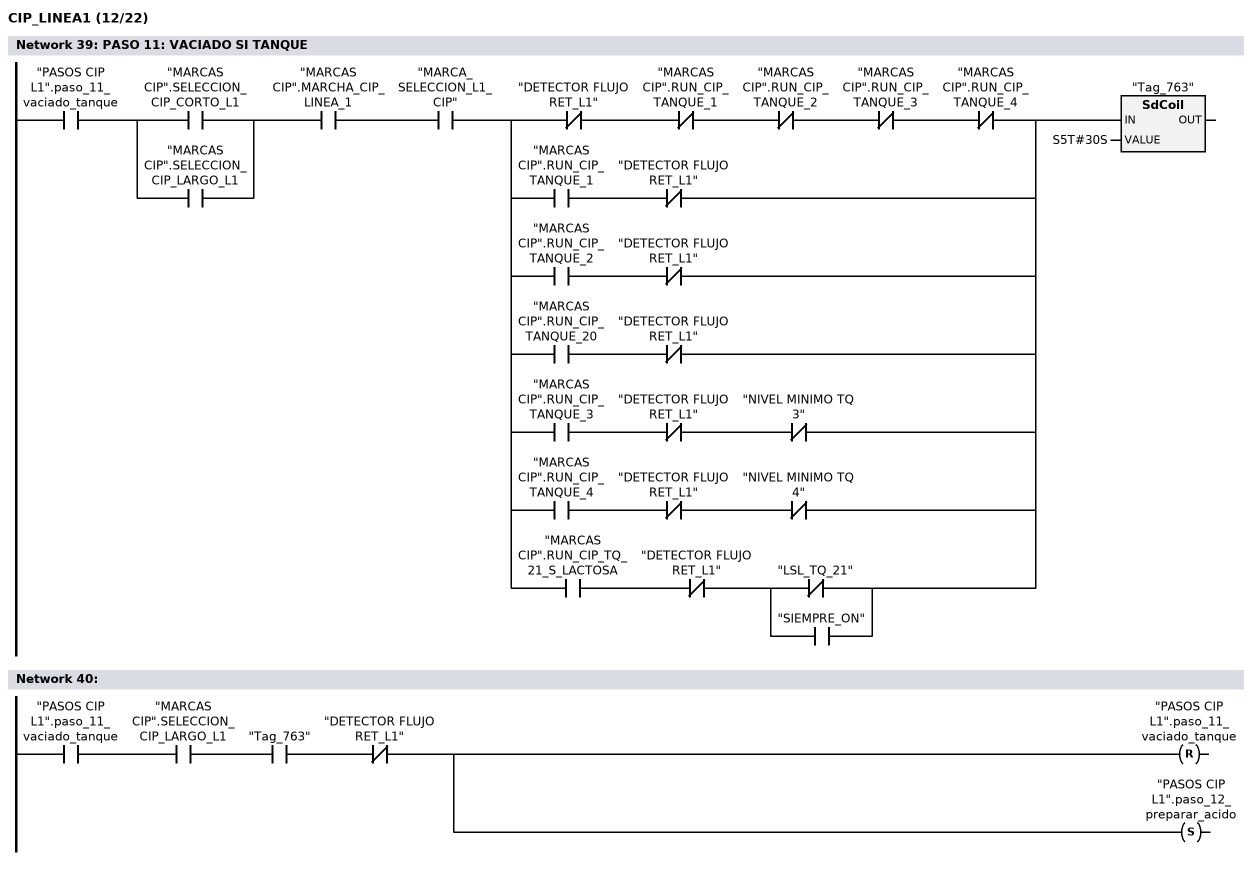
   // no SCL statement known for SdCoil: written as a call
   SdCoil(value := S5T#30S,
          in := "PASOS CIP L1".paso_11_vaciado_tanque AND ("MARCAS CIP".SELECCION_CIP_CORTO_L1 OR "MARCAS CIP".SELECCION_CIP_LARGO_L1) AND "MARCAS CIP".MARCHA_CIP_LINEA_1 AND "MARCA_SELECCION_L1_CIP" AND ((NOT "DETECTOR FLUJO RET_L1" AND NOT "MARCAS CIP".RUN_CIP_TANQUE_1 AND NOT "MARCAS CIP".RUN_CIP_TANQUE_2 AND NOT "MARCAS CIP".RUN_CIP_TANQUE_3 AND NOT "MARCAS CIP".RUN_CIP_TANQUE_4) OR ("MARCAS CIP".RUN_CIP_TANQUE_1 AND NOT "DETECTOR FLUJO RET_L1") OR ("MARCAS CIP".RUN_CIP_TANQUE_2 AND NOT "DETECTOR FLUJO RET_L1") OR ("MARCAS CIP".RUN_CIP_TANQUE_20 AND NOT "DETECTOR FLUJO RET_L1") OR ("MARCAS CIP".RUN_CIP_TANQUE_3 AND NOT "DETECTOR FLUJO RET_L1" AND NOT "NIVEL MINIMO TQ 3") OR ("MARCAS CIP".RUN_CIP_TANQUE_4 AND NOT "DETECTOR FLUJO RET_L1" AND NOT "NIVEL MINIMO TQ 4") OR ("MARCAS CIP".RUN_CIP_TQ_21_S_LACTOSA AND NOT "DETECTOR FLUJO RET_L1" AND (NOT "LSL_TQ_21" OR "SIEMPRE_ON"))),
          operand := "Tag_763");
END_REGION

REGION Network 40
   RUNG wire#powerrail
      Contact( "PASOS CIP L1".paso_11_vaciado_tanque )
      Contact( "MARCAS CIP".SELECCION_CIP_LARGO_L1 )
      Contact( "Tag_763" )
      I_Contact( "DETECTOR FLUJO RET_L1" )
      wire#w1
      R_Coil( "PASOS CIP L1".paso_11_vaciado_tanque )
   END_RUNG
   RUNG wire#w1
      S_Coil( "PASOS CIP L1".paso_12_preparar_acido )
   END_RUNG
   // the same network as SCL:
   #_w1 := "PASOS CIP L1".paso_11_vaciado_tanque AND "MARCAS CIP".SELECCION_CIP_LARGO_L1 AND "Tag_763" AND NOT "DETECTOR FLUJO RET_L1";
   IF #_w1 THEN
       "PASOS CIP L1".paso_11_vaciado_tanque := FALSE;
       "PASOS CIP L1".paso_12_preparar_acido := TRUE;
   END_IF;
END_REGION

REGION Network 41
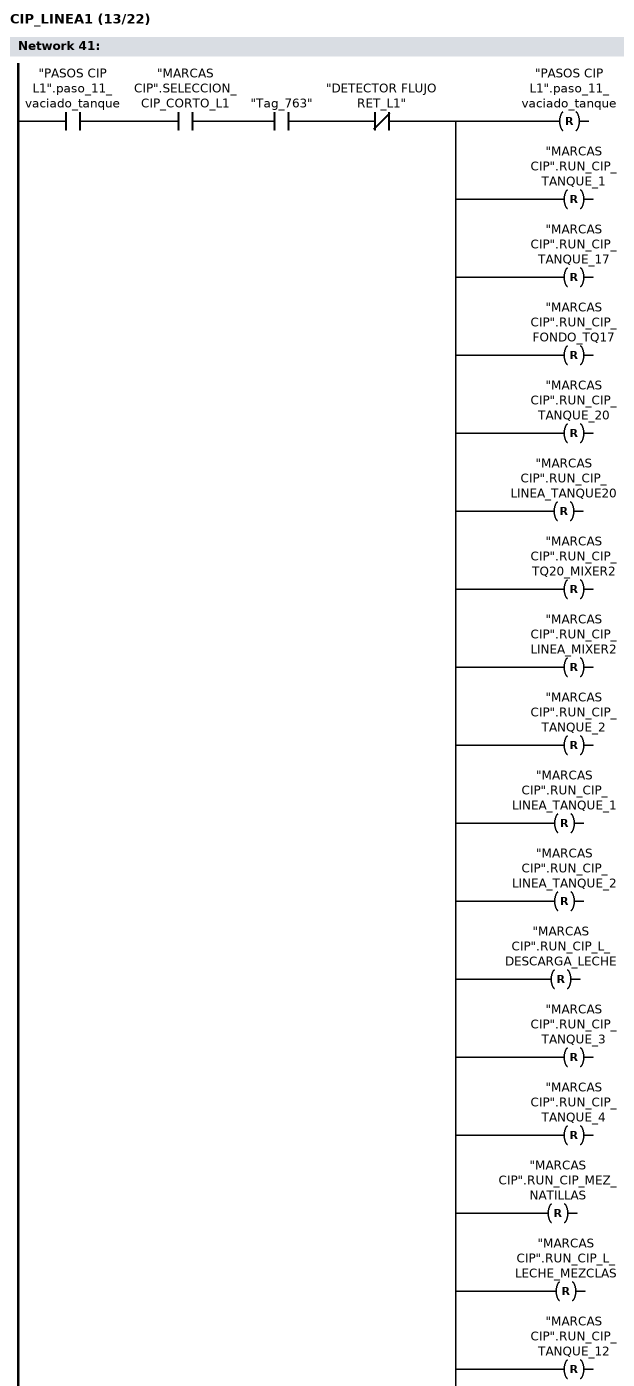
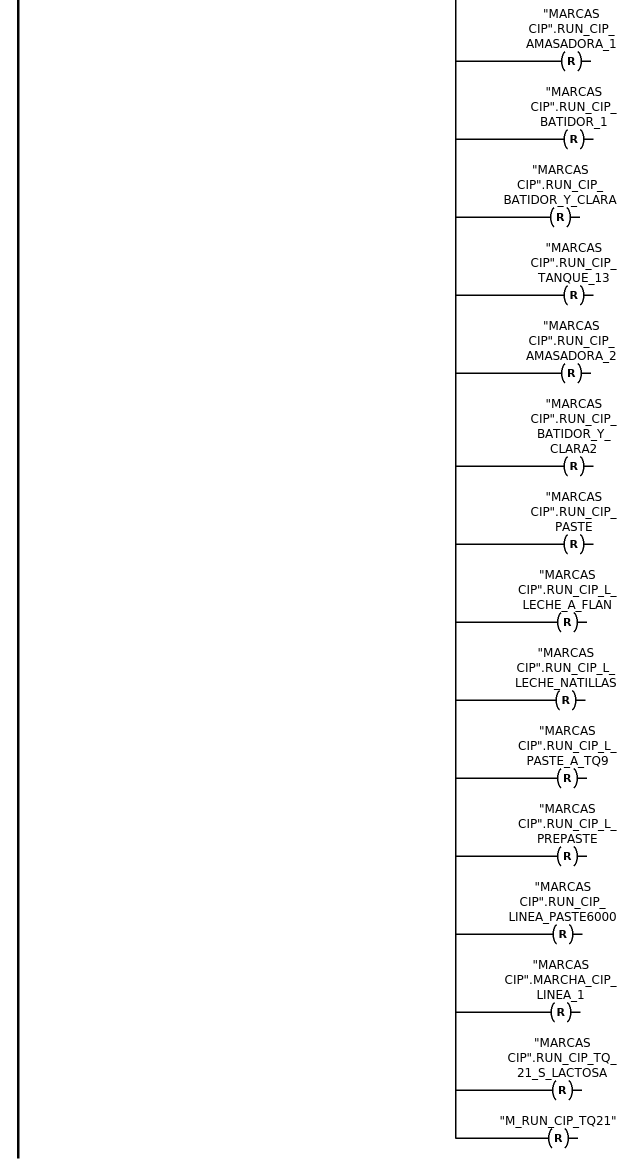
   RUNG wire#powerrail
      Contact( "PASOS CIP L1".paso_11_vaciado_tanque )
      Contact( "MARCAS CIP".SELECCION_CIP_CORTO_L1 )
      Contact( "Tag_763" )
      I_Contact( "DETECTOR FLUJO RET_L1" )
      wire#w1
      R_Coil( "PASOS CIP L1".paso_11_vaciado_tanque )
   END_RUNG
   RUNG wire#w1
      R_Coil( "MARCAS CIP".RUN_CIP_TANQUE_1 )
   END_RUNG
   RUNG wire#w1
      R_Coil( "MARCAS CIP".RUN_CIP_TANQUE_17 )
   END_RUNG
   RUNG wire#w1
      R_Coil( "MARCAS CIP".RUN_CIP_FONDO_TQ17 )
   END_RUNG
   RUNG wire#w1
      R_Coil( "MARCAS CIP".RUN_CIP_TANQUE_20 )
   END_RUNG
   RUNG wire#w1
      R_Coil( "MARCAS CIP".RUN_CIP_LINEA_TANQUE20 )
   END_RUNG
   RUNG wire#w1
      R_Coil( "MARCAS CIP".RUN_CIP_TQ20_MIXER2 )
   END_RUNG
   RUNG wire#w1
      R_Coil( "MARCAS CIP".RUN_CIP_LINEA_MIXER2 )
   END_RUNG
   RUNG wire#w1
      R_Coil( "MARCAS CIP".RUN_CIP_TANQUE_2 )
   END_RUNG
   RUNG wire#w1
      R_Coil( "MARCAS CIP".RUN_CIP_LINEA_TANQUE_1 )
   END_RUNG
   RUNG wire#w1
      R_Coil( "MARCAS CIP".RUN_CIP_LINEA_TANQUE_2 )
   END_RUNG
   RUNG wire#w1
      R_Coil( "MARCAS CIP".RUN_CIP_L_DESCARGA_LECHE )
   END_RUNG
   RUNG wire#w1
      R_Coil( "MARCAS CIP".RUN_CIP_TANQUE_3 )
   END_RUNG
   RUNG wire#w1
      R_Coil( "MARCAS CIP".RUN_CIP_TANQUE_4 )
   END_RUNG
   RUNG wire#w1
      R_Coil( "MARCAS CIP".RUN_CIP_MEZ_NATILLAS )
   END_RUNG
   RUNG wire#w1
      R_Coil( "MARCAS CIP".RUN_CIP_L_LECHE_MEZCLAS )
   END_RUNG
   RUNG wire#w1
      R_Coil( "MARCAS CIP".RUN_CIP_TANQUE_12 )
   END_RUNG
   RUNG wire#w1
      R_Coil( "MARCAS CIP".RUN_CIP_AMASADORA_1 )
   END_RUNG
   RUNG wire#w1
      R_Coil( "MARCAS CIP".RUN_CIP_BATIDOR_1 )
   END_RUNG
   RUNG wire#w1
      R_Coil( "MARCAS CIP".RUN_CIP_BATIDOR_Y_CLARA )
   END_RUNG
   RUNG wire#w1
      R_Coil( "MARCAS CIP".RUN_CIP_TANQUE_13 )
   END_RUNG
   RUNG wire#w1
      R_Coil( "MARCAS CIP".RUN_CIP_AMASADORA_2 )
   END_RUNG
   RUNG wire#w1
      R_Coil( "MARCAS CIP".RUN_CIP_BATIDOR_Y_CLARA2 )
   END_RUNG
   RUNG wire#w1
      R_Coil( "MARCAS CIP".RUN_CIP_PASTE )
   END_RUNG
   RUNG wire#w1
      R_Coil( "MARCAS CIP".RUN_CIP_L_LECHE_A_FLAN )
   END_RUNG
   RUNG wire#w1
      R_Coil( "MARCAS CIP".RUN_CIP_L_LECHE_NATILLAS )
   END_RUNG
   RUNG wire#w1
      R_Coil( "MARCAS CIP".RUN_CIP_L_PASTE_A_TQ9 )
   END_RUNG
   RUNG wire#w1
      R_Coil( "MARCAS CIP".RUN_CIP_L_PREPASTE )
   END_RUNG
   RUNG wire#w1
      R_Coil( "MARCAS CIP".RUN_CIP_LINEA_PASTE6000 )
   END_RUNG
   RUNG wire#w1
      R_Coil( "MARCAS CIP".MARCHA_CIP_LINEA_1 )
   END_RUNG
   RUNG wire#w1
      R_Coil( "MARCAS CIP".RUN_CIP_TQ_21_S_LACTOSA )
   END_RUNG
   RUNG wire#w1
      R_Coil( "M_RUN_CIP_TQ21" )
   END_RUNG
   // the same network as SCL:
   #_w1 := "PASOS CIP L1".paso_11_vaciado_tanque AND "MARCAS CIP".SELECCION_CIP_CORTO_L1 AND "Tag_763" AND NOT "DETECTOR FLUJO RET_L1";
   IF #_w1 THEN
       "PASOS CIP L1".paso_11_vaciado_tanque := FALSE;
       "MARCAS CIP".RUN_CIP_TANQUE_1 := FALSE;
       "MARCAS CIP".RUN_CIP_TANQUE_17 := FALSE;
       "MARCAS CIP".RUN_CIP_FONDO_TQ17 := FALSE;
       "MARCAS CIP".RUN_CIP_TANQUE_20 := FALSE;
       "MARCAS CIP".RUN_CIP_LINEA_TANQUE20 := FALSE;
       "MARCAS CIP".RUN_CIP_TQ20_MIXER2 := FALSE;
       "MARCAS CIP".RUN_CIP_LINEA_MIXER2 := FALSE;
       "MARCAS CIP".RUN_CIP_TANQUE_2 := FALSE;
       "MARCAS CIP".RUN_CIP_LINEA_TANQUE_1 := FALSE;
       "MARCAS CIP".RUN_CIP_LINEA_TANQUE_2 := FALSE;
       "MARCAS CIP".RUN_CIP_L_DESCARGA_LECHE := FALSE;
       "MARCAS CIP".RUN_CIP_TANQUE_3 := FALSE;
       "MARCAS CIP".RUN_CIP_TANQUE_4 := FALSE;
       "MARCAS CIP".RUN_CIP_MEZ_NATILLAS := FALSE;
       "MARCAS CIP".RUN_CIP_L_LECHE_MEZCLAS := FALSE;
       "MARCAS CIP".RUN_CIP_TANQUE_12 := FALSE;
       "MARCAS CIP".RUN_CIP_AMASADORA_1 := FALSE;
       "MARCAS CIP".RUN_CIP_BATIDOR_1 := FALSE;
       "MARCAS CIP".RUN_CIP_BATIDOR_Y_CLARA := FALSE;
       "MARCAS CIP".RUN_CIP_TANQUE_13 := FALSE;
       "MARCAS CIP".RUN_CIP_AMASADORA_2 := FALSE;
       "MARCAS CIP".RUN_CIP_BATIDOR_Y_CLARA2 := FALSE;
       "MARCAS CIP".RUN_CIP_PASTE := FALSE;
       "MARCAS CIP".RUN_CIP_L_LECHE_A_FLAN := FALSE;
       "MARCAS CIP".RUN_CIP_L_LECHE_NATILLAS := FALSE;
       "MARCAS CIP".RUN_CIP_L_PASTE_A_TQ9 := FALSE;
       "MARCAS CIP".RUN_CIP_L_PREPASTE := FALSE;
       "MARCAS CIP".RUN_CIP_LINEA_PASTE6000 := FALSE;
       "MARCAS CIP".MARCHA_CIP_LINEA_1 := FALSE;
       "MARCAS CIP".RUN_CIP_TQ_21_S_LACTOSA := FALSE;
       "M_RUN_CIP_TQ21" := FALSE;
   END_IF;
END_REGION

REGION Network 42
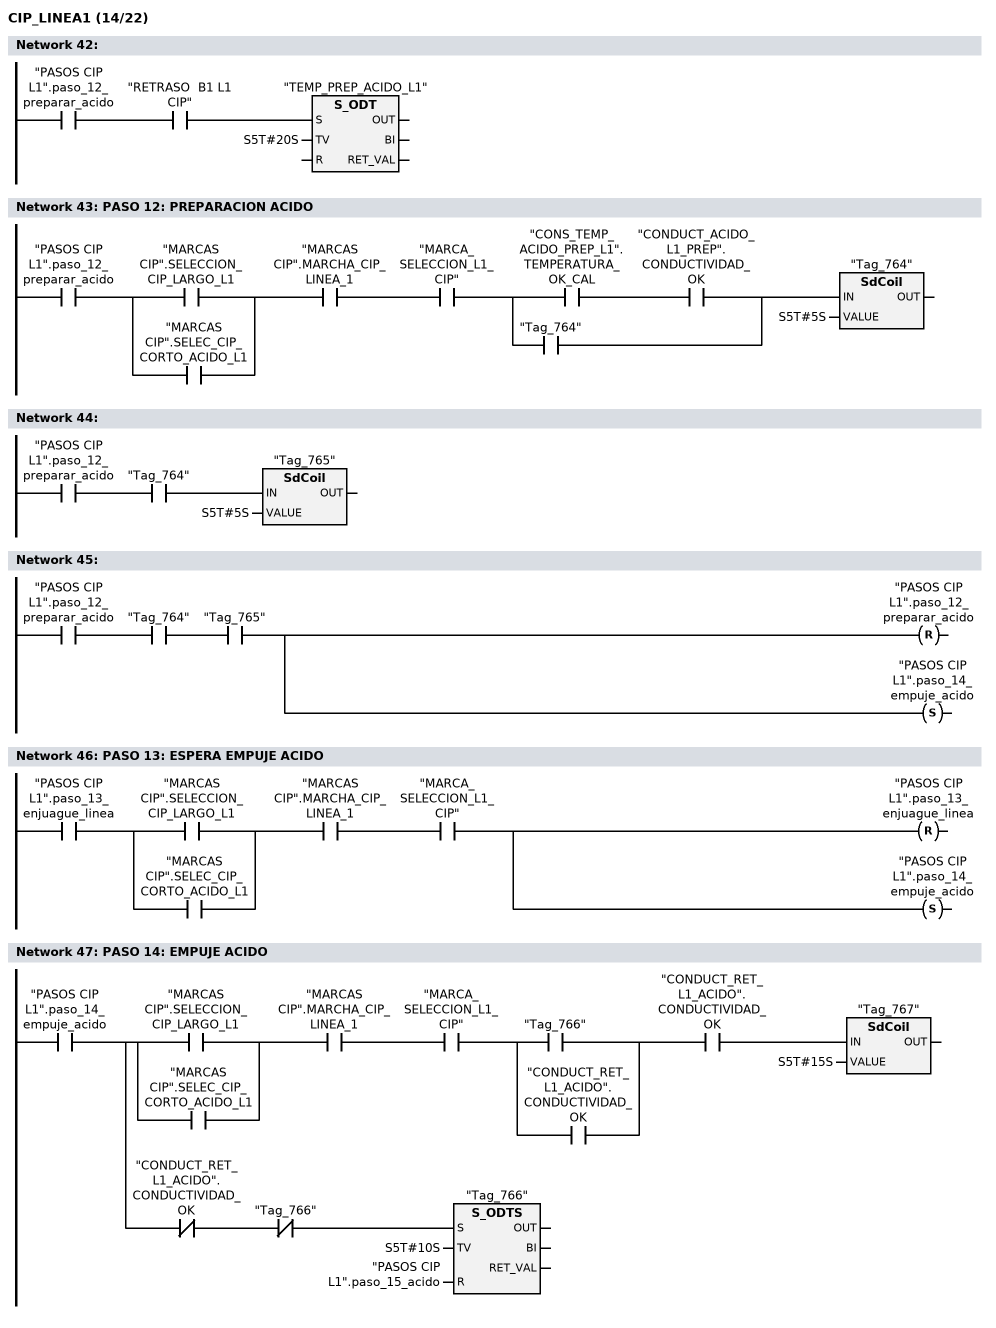
   RUNG wire#powerrail
      Contact( "PASOS CIP L1".paso_12_preparar_acido )
      Contact( "RETRASO  B1 L1 CIP" )
      S_ODT(T_NO := "TEMP_PREP_ACIDO_L1", TV := S5T#20S, R :=, BI =>, RET_VAL =>)
   END_RUNG
   // the same network as SCL:
   #_s5time1 := S_ODT(T_NO := "TEMP_PREP_ACIDO_L1",
                      TV := S5T#20S,
                      S := "PASOS CIP L1".paso_12_preparar_acido AND "RETRASO  B1 L1 CIP");
END_REGION

REGION Network 43: PASO 12: PREPARACION ACIDO
   // no SCL statement known for SdCoil: written as a call
   SdCoil(value := S5T#5S,
          in := "PASOS CIP L1".paso_12_preparar_acido AND ("MARCAS CIP".SELECCION_CIP_LARGO_L1 OR "MARCAS CIP".SELEC_CIP_CORTO_ACIDO_L1) AND "MARCAS CIP".MARCHA_CIP_LINEA_1 AND "MARCA_SELECCION_L1_CIP" AND (("CONS_TEMP_ACIDO_PREP_L1".TEMPERATURA_OK_CAL AND "CONDUCT_ACIDO_L1_PREP".CONDUCTIVIDAD_OK) OR "Tag_764"),
          operand := "Tag_764");
END_REGION

REGION Network 44
   // no SCL statement known for SdCoil: written as a call
   SdCoil(value := S5T#5S, operand := "Tag_765", in := "PASOS CIP L1".paso_12_preparar_acido AND "Tag_764");
END_REGION

REGION Network 45
   RUNG wire#powerrail
      Contact( "PASOS CIP L1".paso_12_preparar_acido )
      Contact( "Tag_764" )
      Contact( "Tag_765" )
      wire#w1
      R_Coil( "PASOS CIP L1".paso_12_preparar_acido )
   END_RUNG
   RUNG wire#w1
      S_Coil( "PASOS CIP L1".paso_14_empuje_acido )
   END_RUNG
   // the same network as SCL:
   #_w1 := "PASOS CIP L1".paso_12_preparar_acido AND "Tag_764" AND "Tag_765";
   IF #_w1 THEN
       "PASOS CIP L1".paso_12_preparar_acido := FALSE;
       "PASOS CIP L1".paso_14_empuje_acido := TRUE;
   END_IF;
END_REGION

REGION Network 46: PASO 13: ESPERA EMPUJE ACIDO
   RUNG wire#powerrail
      Contact( "PASOS CIP L1".paso_13_enjuague_linea )
      wire#w1
      Contact( "MARCAS CIP".SELECCION_CIP_LARGO_L1 )
      wire#w2
      Contact( "MARCAS CIP".MARCHA_CIP_LINEA_1 )
      Contact( "MARCA_SELECCION_L1_CIP" )
      wire#w3
      R_Coil( "PASOS CIP L1".paso_13_enjuague_linea )
   END_RUNG
   RUNG wire#w1
      Contact( "MARCAS CIP".SELEC_CIP_CORTO_ACIDO_L1 )
   END_RUNG wire#w2
   RUNG wire#w3
      S_Coil( "PASOS CIP L1".paso_14_empuje_acido )
   END_RUNG
   // the same network as SCL:
   #_w1 := "PASOS CIP L1".paso_13_enjuague_linea AND ("MARCAS CIP".SELECCION_CIP_LARGO_L1 OR "MARCAS CIP".SELEC_CIP_CORTO_ACIDO_L1) AND "MARCAS CIP".MARCHA_CIP_LINEA_1 AND "MARCA_SELECCION_L1_CIP";
   IF #_w1 THEN
       "PASOS CIP L1".paso_13_enjuague_linea := FALSE;
       "PASOS CIP L1".paso_14_empuje_acido := TRUE;
   END_IF;
END_REGION

REGION Network 47: PASO 14: EMPUJE ACIDO
   // no SCL statement known for SdCoil: written as a call
   #_w1 := "PASOS CIP L1".paso_14_empuje_acido;
   SdCoil(value := S5T#15S,
          operand := "Tag_767",
          in := "PASOS CIP L1".paso_14_empuje_acido AND ("MARCAS CIP".SELECCION_CIP_LARGO_L1 OR "MARCAS CIP".SELEC_CIP_CORTO_ACIDO_L1) AND "MARCAS CIP".MARCHA_CIP_LINEA_1 AND "MARCA_SELECCION_L1_CIP" AND ("Tag_766" OR "CONDUCT_RET_L1_ACIDO".CONDUCTIVIDAD_OK) AND "CONDUCT_RET_L1_ACIDO".CONDUCTIVIDAD_OK);
   #_s5time1 := S_ODTS(T_NO := "Tag_766",
                       TV := S5T#10S,
                       R := "PASOS CIP L1".paso_15_acido,
                       S := #_w1 AND NOT "CONDUCT_RET_L1_ACIDO".CONDUCTIVIDAD_OK AND NOT "Tag_766");
END_REGION

REGION Network 48
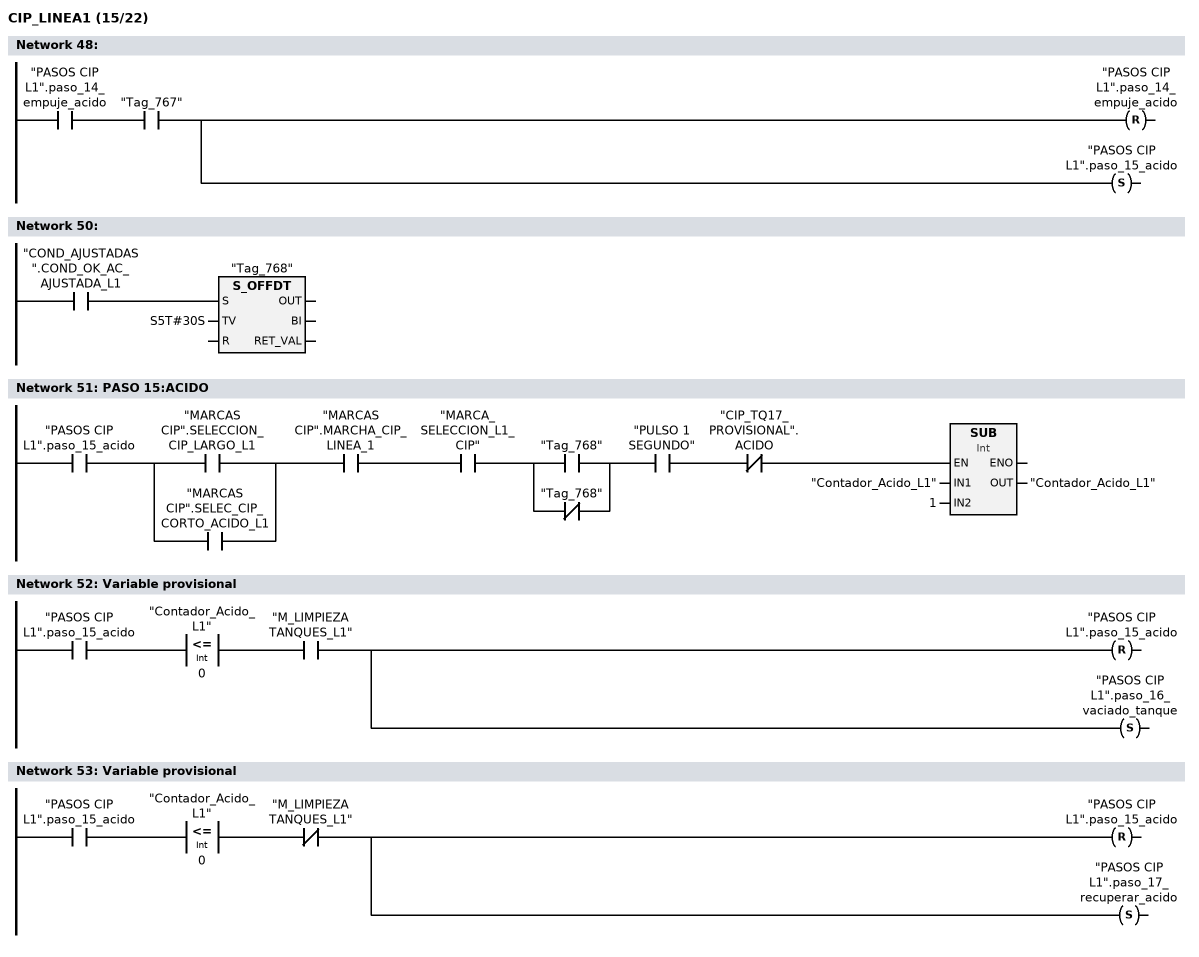
   RUNG wire#powerrail
      Contact( "PASOS CIP L1".paso_14_empuje_acido )
      Contact( "Tag_767" )
      wire#w1
      R_Coil( "PASOS CIP L1".paso_14_empuje_acido )
   END_RUNG
   RUNG wire#w1
      S_Coil( "PASOS CIP L1".paso_15_acido )
   END_RUNG
   // the same network as SCL:
   #_w1 := "PASOS CIP L1".paso_14_empuje_acido AND "Tag_767";
   IF #_w1 THEN
       "PASOS CIP L1".paso_14_empuje_acido := FALSE;
       "PASOS CIP L1".paso_15_acido := TRUE;
   END_IF;
END_REGION

NETWORK
TITLE = 
      A     "PASOS CIP L1".paso_15_acido;
      JC    c2;
      L     "SP TIM L1 CIP".TIM_PASO_15_L1;
      L     60;
      *I;
      T     "Contador_Acido_L1";
c2:   NOP   0;

REGION Network 50
   RUNG wire#powerrail
      Contact( "COND_AJUSTADAS".COND_OK_AC_AJUSTADA_L1 )
      S_OFFDT(T_NO := "Tag_768", TV := S5T#30S, R :=, BI =>, RET_VAL =>)
   END_RUNG
   // the same network as SCL:
   #_s5time1 := S_OFFDT(T_NO := "Tag_768", TV := S5T#30S, S := "COND_AJUSTADAS".COND_OK_AC_AJUSTADA_L1);
END_REGION

REGION Network 51: PASO 15:ACIDO
   RUNG wire#powerrail
      Contact( "PASOS CIP L1".paso_15_acido )
      wire#w1
      Contact( "MARCAS CIP".SELECCION_CIP_LARGO_L1 )
      wire#w2
      Contact( "MARCAS CIP".MARCHA_CIP_LINEA_1 )
      Contact( "MARCA_SELECCION_L1_CIP" )
      wire#w3
      Contact( "Tag_768" )
      wire#w4
      Contact( "PULSO 1 SEGUNDO" )
      I_Contact( "CIP_TQ17_PROVISIONAL".ACIDO )
      { S7_Templates := "SrcType := Int"; S7_GenerateENO := "TRUE" } Sub(in1 := "Contador_Acido_L1", in2 := 1, out => "Contador_Acido_L1")
   END_RUNG
   RUNG wire#w1
      Contact( "MARCAS CIP".SELEC_CIP_CORTO_ACIDO_L1 )
   END_RUNG wire#w2
   RUNG wire#w3
      I_Contact( "Tag_768" )
   END_RUNG wire#w4
   // the same network as SCL:
   IF "PASOS CIP L1".paso_15_acido AND ("MARCAS CIP".SELECCION_CIP_LARGO_L1 OR "MARCAS CIP".SELEC_CIP_CORTO_ACIDO_L1) AND "MARCAS CIP".MARCHA_CIP_LINEA_1 AND "MARCA_SELECCION_L1_CIP" AND ("Tag_768" OR NOT "Tag_768") AND "PULSO 1 SEGUNDO" AND NOT "CIP_TQ17_PROVISIONAL".ACIDO THEN
       "Contador_Acido_L1" := "Contador_Acido_L1" - 1;
   END_IF;
END_REGION

REGION Network 52: Variable provisional
   RUNG wire#powerrail
      Contact( "PASOS CIP L1".paso_15_acido )
      { S7_Templates := "SrcType := Int" } LE_Contact(in1 := "Contador_Acido_L1", in2 := 0)
      Contact( "M_LIMPIEZA TANQUES_L1" )
      wire#w1
      R_Coil( "PASOS CIP L1".paso_15_acido )
   END_RUNG
   RUNG wire#w1
      S_Coil( "PASOS CIP L1".paso_16_vaciado_tanque )
   END_RUNG
   // the same network as SCL:
   #_w1 := "PASOS CIP L1".paso_15_acido AND ("Contador_Acido_L1" <= 0) AND "M_LIMPIEZA TANQUES_L1";
   IF #_w1 THEN
       "PASOS CIP L1".paso_15_acido := FALSE;
       "PASOS CIP L1".paso_16_vaciado_tanque := TRUE;
   END_IF;
END_REGION

REGION Network 53: Variable provisional
   RUNG wire#powerrail
      Contact( "PASOS CIP L1".paso_15_acido )
      { S7_Templates := "SrcType := Int" } LE_Contact(in1 := "Contador_Acido_L1", in2 := 0)
      I_Contact( "M_LIMPIEZA TANQUES_L1" )
      wire#w1
      R_Coil( "PASOS CIP L1".paso_15_acido )
   END_RUNG
   RUNG wire#w1
      S_Coil( "PASOS CIP L1".paso_17_recuperar_acido )
   END_RUNG
   // the same network as SCL:
   #_w1 := "PASOS CIP L1".paso_15_acido AND ("Contador_Acido_L1" <= 0) AND NOT "M_LIMPIEZA TANQUES_L1";
   IF #_w1 THEN
       "PASOS CIP L1".paso_15_acido := FALSE;
       "PASOS CIP L1".paso_17_recuperar_acido := TRUE;
   END_IF;
END_REGION

REGION Network 54: PASO 16: VACIADO SI TANQUES
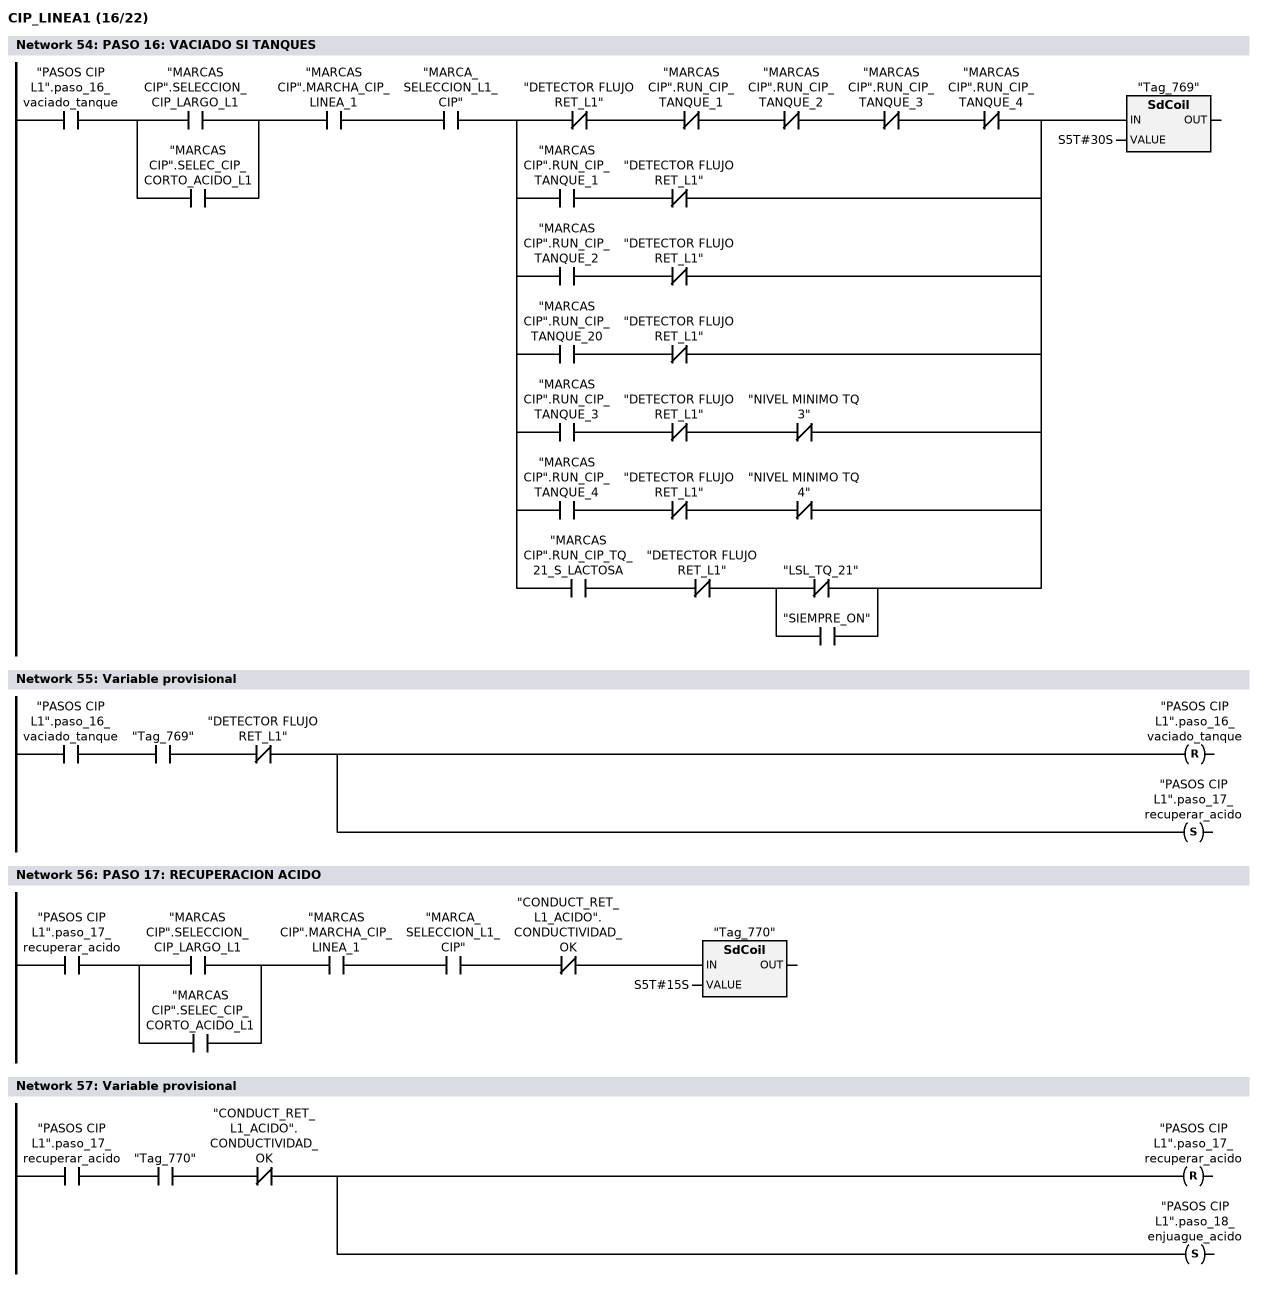
   // no SCL statement known for SdCoil: written as a call
   SdCoil(value := S5T#30S,
          in := "PASOS CIP L1".paso_16_vaciado_tanque AND ("MARCAS CIP".SELECCION_CIP_LARGO_L1 OR "MARCAS CIP".SELEC_CIP_CORTO_ACIDO_L1) AND "MARCAS CIP".MARCHA_CIP_LINEA_1 AND "MARCA_SELECCION_L1_CIP" AND ((NOT "DETECTOR FLUJO RET_L1" AND NOT "MARCAS CIP".RUN_CIP_TANQUE_1 AND NOT "MARCAS CIP".RUN_CIP_TANQUE_2 AND NOT "MARCAS CIP".RUN_CIP_TANQUE_3 AND NOT "MARCAS CIP".RUN_CIP_TANQUE_4) OR ("MARCAS CIP".RUN_CIP_TANQUE_1 AND NOT "DETECTOR FLUJO RET_L1") OR ("MARCAS CIP".RUN_CIP_TANQUE_2 AND NOT "DETECTOR FLUJO RET_L1") OR ("MARCAS CIP".RUN_CIP_TANQUE_20 AND NOT "DETECTOR FLUJO RET_L1") OR ("MARCAS CIP".RUN_CIP_TANQUE_3 AND NOT "DETECTOR FLUJO RET_L1" AND NOT "NIVEL MINIMO TQ 3") OR ("MARCAS CIP".RUN_CIP_TANQUE_4 AND NOT "DETECTOR FLUJO RET_L1" AND NOT "NIVEL MINIMO TQ 4") OR ("MARCAS CIP".RUN_CIP_TQ_21_S_LACTOSA AND NOT "DETECTOR FLUJO RET_L1" AND (NOT "LSL_TQ_21" OR "SIEMPRE_ON"))),
          operand := "Tag_769");
END_REGION

REGION Network 55: Variable provisional
   RUNG wire#powerrail
      Contact( "PASOS CIP L1".paso_16_vaciado_tanque )
      Contact( "Tag_769" )
      I_Contact( "DETECTOR FLUJO RET_L1" )
      wire#w1
      R_Coil( "PASOS CIP L1".paso_16_vaciado_tanque )
   END_RUNG
   RUNG wire#w1
      S_Coil( "PASOS CIP L1".paso_17_recuperar_acido )
   END_RUNG
   // the same network as SCL:
   #_w1 := "PASOS CIP L1".paso_16_vaciado_tanque AND "Tag_769" AND NOT "DETECTOR FLUJO RET_L1";
   IF #_w1 THEN
       "PASOS CIP L1".paso_16_vaciado_tanque := FALSE;
       "PASOS CIP L1".paso_17_recuperar_acido := TRUE;
   END_IF;
END_REGION

REGION Network 56: PASO 17: RECUPERACION ACIDO
   // no SCL statement known for SdCoil: written as a call
   SdCoil(value := S5T#15S,
          operand := "Tag_770",
          in := "PASOS CIP L1".paso_17_recuperar_acido AND ("MARCAS CIP".SELECCION_CIP_LARGO_L1 OR "MARCAS CIP".SELEC_CIP_CORTO_ACIDO_L1) AND "MARCAS CIP".MARCHA_CIP_LINEA_1 AND "MARCA_SELECCION_L1_CIP" AND NOT "CONDUCT_RET_L1_ACIDO".CONDUCTIVIDAD_OK);
END_REGION

REGION Network 57: Variable provisional
   RUNG wire#powerrail
      Contact( "PASOS CIP L1".paso_17_recuperar_acido )
      Contact( "Tag_770" )
      I_Contact( "CONDUCT_RET_L1_ACIDO".CONDUCTIVIDAD_OK )
      wire#w1
      R_Coil( "PASOS CIP L1".paso_17_recuperar_acido )
   END_RUNG
   RUNG wire#w1
      S_Coil( "PASOS CIP L1".paso_18_enjuague_acido )
   END_RUNG
   // the same network as SCL:
   #_w1 := "PASOS CIP L1".paso_17_recuperar_acido AND "Tag_770" AND NOT "CONDUCT_RET_L1_ACIDO".CONDUCTIVIDAD_OK;
   IF #_w1 THEN
       "PASOS CIP L1".paso_17_recuperar_acido := FALSE;
       "PASOS CIP L1".paso_18_enjuague_acido := TRUE;
   END_IF;
END_REGION

REGION Network 58: PASO 18: ENJUAGUE ACIDO
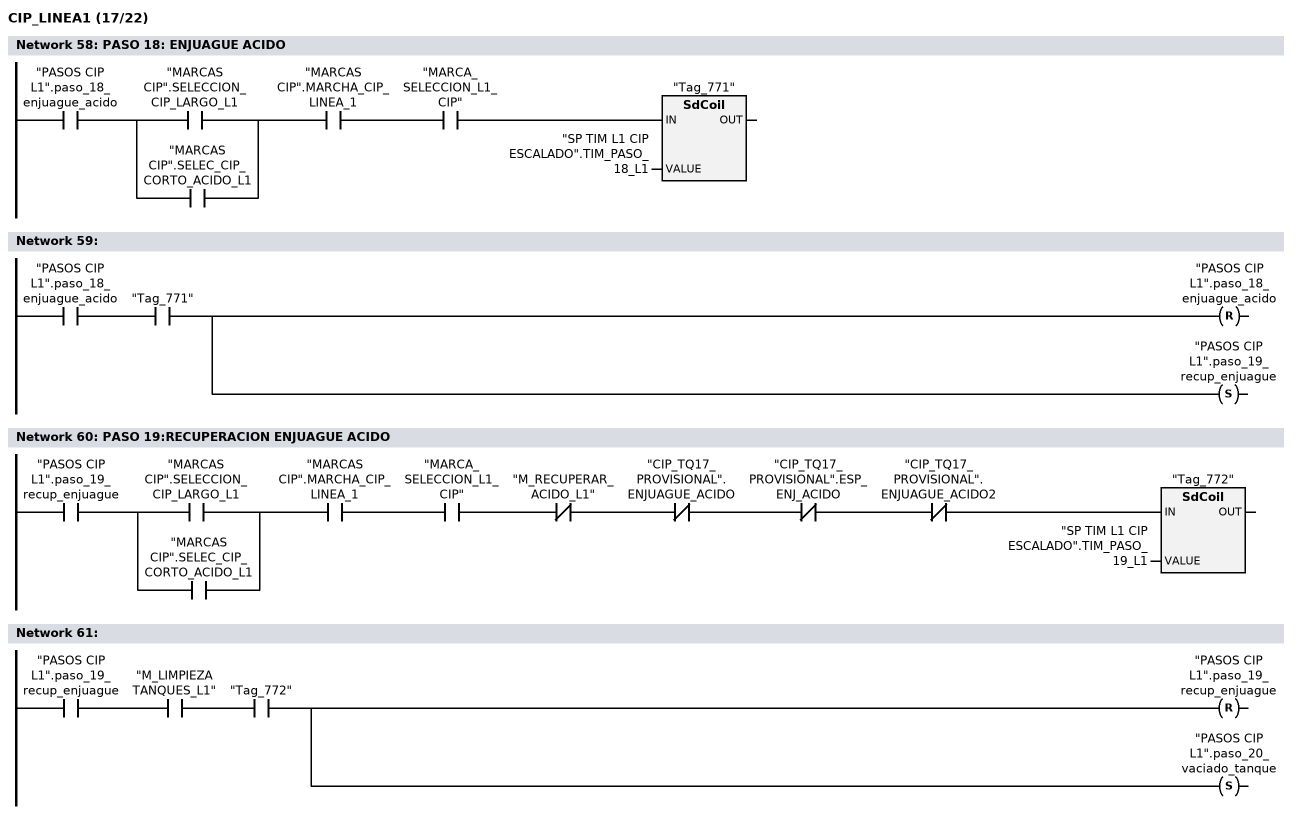
   // no SCL statement known for SdCoil: written as a call
   SdCoil(value := "SP TIM L1 CIP ESCALADO".TIM_PASO_18_L1,
          operand := "Tag_771",
          in := "PASOS CIP L1".paso_18_enjuague_acido AND ("MARCAS CIP".SELECCION_CIP_LARGO_L1 OR "MARCAS CIP".SELEC_CIP_CORTO_ACIDO_L1) AND "MARCAS CIP".MARCHA_CIP_LINEA_1 AND "MARCA_SELECCION_L1_CIP");
END_REGION

REGION Network 59
   RUNG wire#powerrail
      Contact( "PASOS CIP L1".paso_18_enjuague_acido )
      Contact( "Tag_771" )
      wire#w1
      R_Coil( "PASOS CIP L1".paso_18_enjuague_acido )
   END_RUNG
   RUNG wire#w1
      S_Coil( "PASOS CIP L1".paso_19_recup_enjuague )
   END_RUNG
   // the same network as SCL:
   #_w1 := "PASOS CIP L1".paso_18_enjuague_acido AND "Tag_771";
   IF #_w1 THEN
       "PASOS CIP L1".paso_18_enjuague_acido := FALSE;
       "PASOS CIP L1".paso_19_recup_enjuague := TRUE;
   END_IF;
END_REGION

REGION Network 60: PASO 19:RECUPERACION ENJUAGUE ACIDO
   // no SCL statement known for SdCoil: written as a call
   SdCoil(value := "SP TIM L1 CIP ESCALADO".TIM_PASO_19_L1,
          operand := "Tag_772",
          in := "PASOS CIP L1".paso_19_recup_enjuague AND ("MARCAS CIP".SELECCION_CIP_LARGO_L1 OR "MARCAS CIP".SELEC_CIP_CORTO_ACIDO_L1) AND "MARCAS CIP".MARCHA_CIP_LINEA_1 AND "MARCA_SELECCION_L1_CIP" AND NOT "M_RECUPERAR_ACIDO_L1" AND NOT "CIP_TQ17_PROVISIONAL".ENJUAGUE_ACIDO AND NOT "CIP_TQ17_PROVISIONAL".ESP_ENJ_ACIDO AND NOT "CIP_TQ17_PROVISIONAL".ENJUAGUE_ACIDO2);
END_REGION

REGION Network 61
   RUNG wire#powerrail
      Contact( "PASOS CIP L1".paso_19_recup_enjuague )
      Contact( "M_LIMPIEZA TANQUES_L1" )
      Contact( "Tag_772" )
      wire#w1
      R_Coil( "PASOS CIP L1".paso_19_recup_enjuague )
   END_RUNG
   RUNG wire#w1
      S_Coil( "PASOS CIP L1".paso_20_vaciado_tanque )
   END_RUNG
   // the same network as SCL:
   #_w1 := "PASOS CIP L1".paso_19_recup_enjuague AND "M_LIMPIEZA TANQUES_L1" AND "Tag_772";
   IF #_w1 THEN
       "PASOS CIP L1".paso_19_recup_enjuague := FALSE;
       "PASOS CIP L1".paso_20_vaciado_tanque := TRUE;
   END_IF;
END_REGION

REGION Network 62
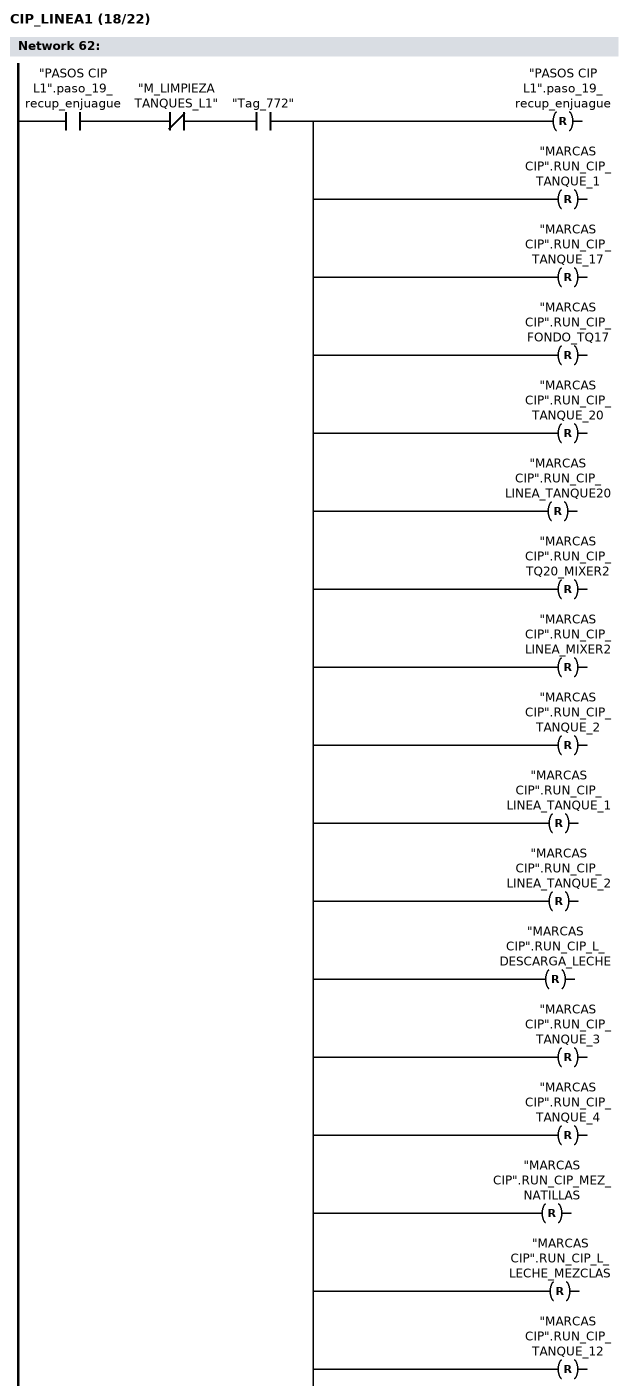
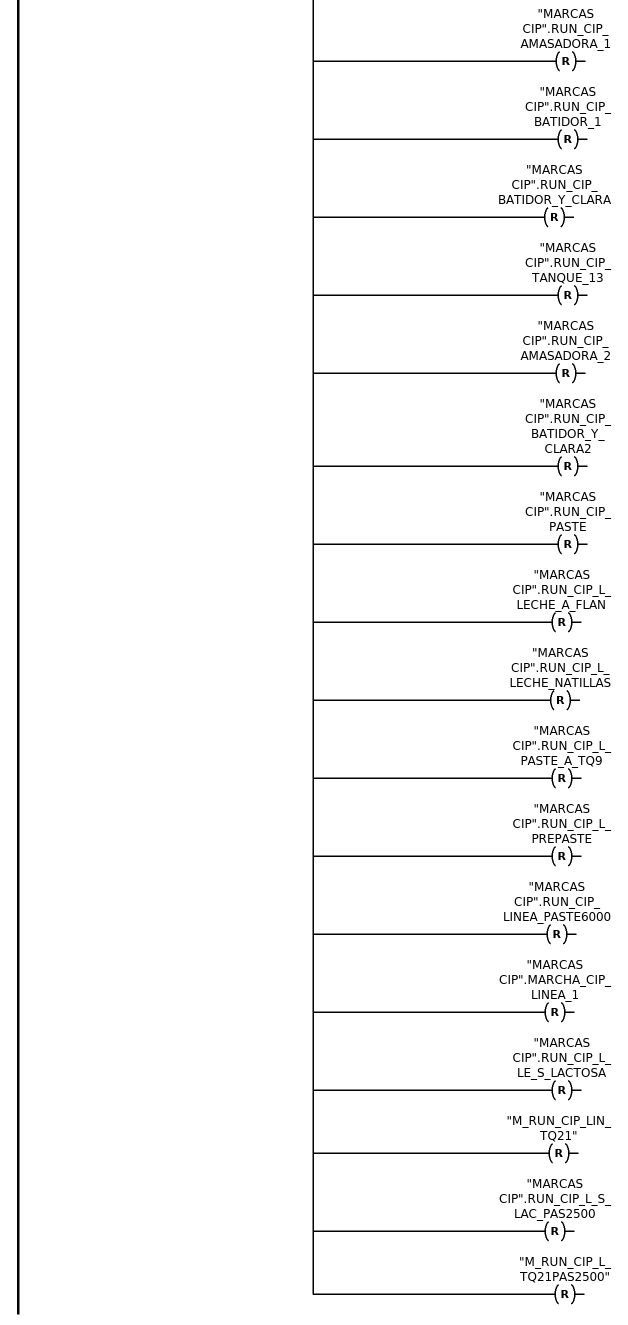
   RUNG wire#powerrail
      Contact( "PASOS CIP L1".paso_19_recup_enjuague )
      I_Contact( "M_LIMPIEZA TANQUES_L1" )
      Contact( "Tag_772" )
      wire#w1
      R_Coil( "PASOS CIP L1".paso_19_recup_enjuague )
   END_RUNG
   RUNG wire#w1
      R_Coil( "MARCAS CIP".RUN_CIP_TANQUE_1 )
   END_RUNG
   RUNG wire#w1
      R_Coil( "MARCAS CIP".RUN_CIP_TANQUE_17 )
   END_RUNG
   RUNG wire#w1
      R_Coil( "MARCAS CIP".RUN_CIP_FONDO_TQ17 )
   END_RUNG
   RUNG wire#w1
      R_Coil( "MARCAS CIP".RUN_CIP_TANQUE_20 )
   END_RUNG
   RUNG wire#w1
      R_Coil( "MARCAS CIP".RUN_CIP_LINEA_TANQUE20 )
   END_RUNG
   RUNG wire#w1
      R_Coil( "MARCAS CIP".RUN_CIP_TQ20_MIXER2 )
   END_RUNG
   RUNG wire#w1
      R_Coil( "MARCAS CIP".RUN_CIP_LINEA_MIXER2 )
   END_RUNG
   RUNG wire#w1
      R_Coil( "MARCAS CIP".RUN_CIP_TANQUE_2 )
   END_RUNG
   RUNG wire#w1
      R_Coil( "MARCAS CIP".RUN_CIP_LINEA_TANQUE_1 )
   END_RUNG
   RUNG wire#w1
      R_Coil( "MARCAS CIP".RUN_CIP_LINEA_TANQUE_2 )
   END_RUNG
   RUNG wire#w1
      R_Coil( "MARCAS CIP".RUN_CIP_L_DESCARGA_LECHE )
   END_RUNG
   RUNG wire#w1
      R_Coil( "MARCAS CIP".RUN_CIP_TANQUE_3 )
   END_RUNG
   RUNG wire#w1
      R_Coil( "MARCAS CIP".RUN_CIP_TANQUE_4 )
   END_RUNG
   RUNG wire#w1
      R_Coil( "MARCAS CIP".RUN_CIP_MEZ_NATILLAS )
   END_RUNG
   RUNG wire#w1
      R_Coil( "MARCAS CIP".RUN_CIP_L_LECHE_MEZCLAS )
   END_RUNG
   RUNG wire#w1
      R_Coil( "MARCAS CIP".RUN_CIP_TANQUE_12 )
   END_RUNG
   RUNG wire#w1
      R_Coil( "MARCAS CIP".RUN_CIP_AMASADORA_1 )
   END_RUNG
   RUNG wire#w1
      R_Coil( "MARCAS CIP".RUN_CIP_BATIDOR_1 )
   END_RUNG
   RUNG wire#w1
      R_Coil( "MARCAS CIP".RUN_CIP_BATIDOR_Y_CLARA )
   END_RUNG
   RUNG wire#w1
      R_Coil( "MARCAS CIP".RUN_CIP_TANQUE_13 )
   END_RUNG
   RUNG wire#w1
      R_Coil( "MARCAS CIP".RUN_CIP_AMASADORA_2 )
   END_RUNG
   RUNG wire#w1
      R_Coil( "MARCAS CIP".RUN_CIP_BATIDOR_Y_CLARA2 )
   END_RUNG
   RUNG wire#w1
      R_Coil( "MARCAS CIP".RUN_CIP_PASTE )
   END_RUNG
   RUNG wire#w1
      R_Coil( "MARCAS CIP".RUN_CIP_L_LECHE_A_FLAN )
   END_RUNG
   RUNG wire#w1
      R_Coil( "MARCAS CIP".RUN_CIP_L_LECHE_NATILLAS )
   END_RUNG
   RUNG wire#w1
      R_Coil( "MARCAS CIP".RUN_CIP_L_PASTE_A_TQ9 )
   END_RUNG
   RUNG wire#w1
      R_Coil( "MARCAS CIP".RUN_CIP_L_PREPASTE )
   END_RUNG
   RUNG wire#w1
      R_Coil( "MARCAS CIP".RUN_CIP_LINEA_PASTE6000 )
   END_RUNG
   RUNG wire#w1
      R_Coil( "MARCAS CIP".MARCHA_CIP_LINEA_1 )
   END_RUNG
   RUNG wire#w1
      R_Coil( "MARCAS CIP".RUN_CIP_L_LE_S_LACTOSA )
   END_RUNG
   RUNG wire#w1
      R_Coil( "M_RUN_CIP_LIN_TQ21" )
   END_RUNG
   RUNG wire#w1
      R_Coil( "MARCAS CIP".RUN_CIP_L_S_LAC_PAS2500 )
   END_RUNG
   RUNG wire#w1
      R_Coil( "M_RUN_CIP_L_TQ21PAS2500" )
   END_RUNG
   // the same network as SCL:
   #_w1 := "PASOS CIP L1".paso_19_recup_enjuague AND NOT "M_LIMPIEZA TANQUES_L1" AND "Tag_772";
   IF #_w1 THEN
       "PASOS CIP L1".paso_19_recup_enjuague := FALSE;
       "MARCAS CIP".RUN_CIP_TANQUE_1 := FALSE;
       "MARCAS CIP".RUN_CIP_TANQUE_17 := FALSE;
       "MARCAS CIP".RUN_CIP_FONDO_TQ17 := FALSE;
       "MARCAS CIP".RUN_CIP_TANQUE_20 := FALSE;
       "MARCAS CIP".RUN_CIP_LINEA_TANQUE20 := FALSE;
       "MARCAS CIP".RUN_CIP_TQ20_MIXER2 := FALSE;
       "MARCAS CIP".RUN_CIP_LINEA_MIXER2 := FALSE;
       "MARCAS CIP".RUN_CIP_TANQUE_2 := FALSE;
       "MARCAS CIP".RUN_CIP_LINEA_TANQUE_1 := FALSE;
       "MARCAS CIP".RUN_CIP_LINEA_TANQUE_2 := FALSE;
       "MARCAS CIP".RUN_CIP_L_DESCARGA_LECHE := FALSE;
       "MARCAS CIP".RUN_CIP_TANQUE_3 := FALSE;
       "MARCAS CIP".RUN_CIP_TANQUE_4 := FALSE;
       "MARCAS CIP".RUN_CIP_MEZ_NATILLAS := FALSE;
       "MARCAS CIP".RUN_CIP_L_LECHE_MEZCLAS := FALSE;
       "MARCAS CIP".RUN_CIP_TANQUE_12 := FALSE;
       "MARCAS CIP".RUN_CIP_AMASADORA_1 := FALSE;
       "MARCAS CIP".RUN_CIP_BATIDOR_1 := FALSE;
       "MARCAS CIP".RUN_CIP_BATIDOR_Y_CLARA := FALSE;
       "MARCAS CIP".RUN_CIP_TANQUE_13 := FALSE;
       "MARCAS CIP".RUN_CIP_AMASADORA_2 := FALSE;
       "MARCAS CIP".RUN_CIP_BATIDOR_Y_CLARA2 := FALSE;
       "MARCAS CIP".RUN_CIP_PASTE := FALSE;
       "MARCAS CIP".RUN_CIP_L_LECHE_A_FLAN := FALSE;
       "MARCAS CIP".RUN_CIP_L_LECHE_NATILLAS := FALSE;
       "MARCAS CIP".RUN_CIP_L_PASTE_A_TQ9 := FALSE;
       "MARCAS CIP".RUN_CIP_L_PREPASTE := FALSE;
       "MARCAS CIP".RUN_CIP_LINEA_PASTE6000 := FALSE;
       "MARCAS CIP".MARCHA_CIP_LINEA_1 := FALSE;
       "MARCAS CIP".RUN_CIP_L_LE_S_LACTOSA := FALSE;
       "M_RUN_CIP_LIN_TQ21" := FALSE;
       "MARCAS CIP".RUN_CIP_L_S_LAC_PAS2500 := FALSE;
       "M_RUN_CIP_L_TQ21PAS2500" := FALSE;
   END_IF;
END_REGION

REGION Network 63: PASO 19: VACIADO SI TANQUES
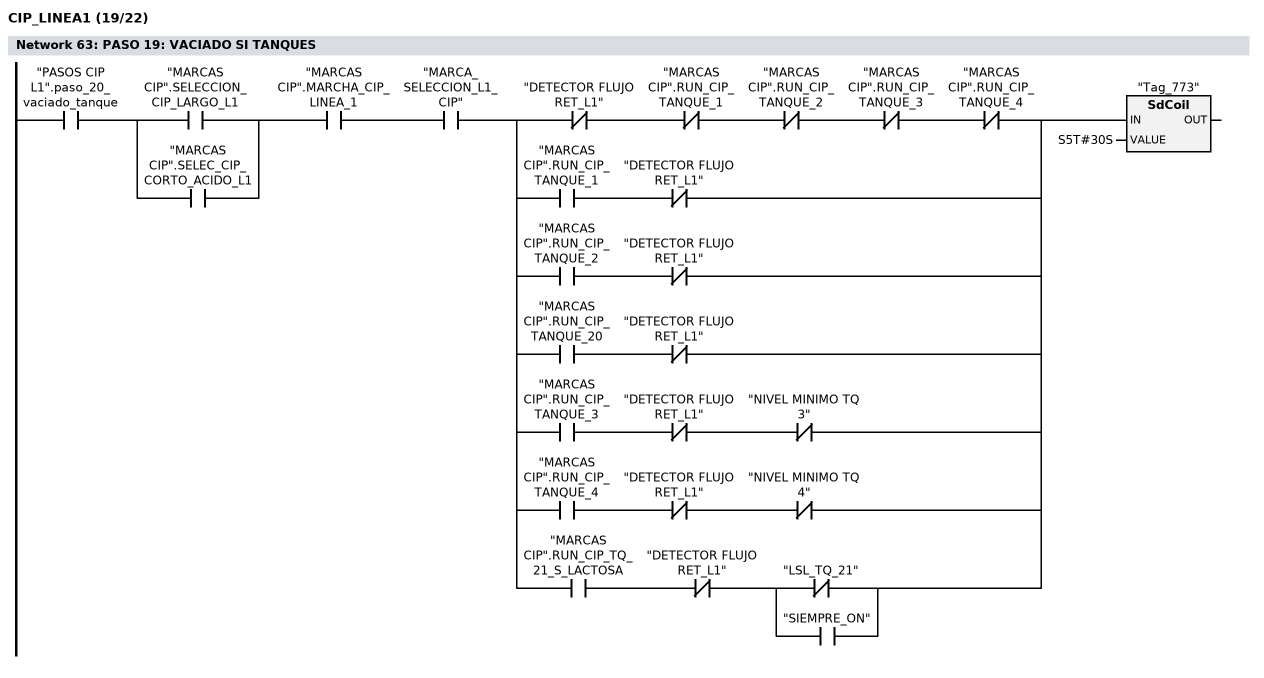
   // no SCL statement known for SdCoil: written as a call
   SdCoil(value := S5T#30S,
          in := "PASOS CIP L1".paso_20_vaciado_tanque AND ("MARCAS CIP".SELECCION_CIP_LARGO_L1 OR "MARCAS CIP".SELEC_CIP_CORTO_ACIDO_L1) AND "MARCAS CIP".MARCHA_CIP_LINEA_1 AND "MARCA_SELECCION_L1_CIP" AND ((NOT "DETECTOR FLUJO RET_L1" AND NOT "MARCAS CIP".RUN_CIP_TANQUE_1 AND NOT "MARCAS CIP".RUN_CIP_TANQUE_2 AND NOT "MARCAS CIP".RUN_CIP_TANQUE_3 AND NOT "MARCAS CIP".RUN_CIP_TANQUE_4) OR ("MARCAS CIP".RUN_CIP_TANQUE_1 AND NOT "DETECTOR FLUJO RET_L1") OR ("MARCAS CIP".RUN_CIP_TANQUE_2 AND NOT "DETECTOR FLUJO RET_L1") OR ("MARCAS CIP".RUN_CIP_TANQUE_20 AND NOT "DETECTOR FLUJO RET_L1") OR ("MARCAS CIP".RUN_CIP_TANQUE_3 AND NOT "DETECTOR FLUJO RET_L1" AND NOT "NIVEL MINIMO TQ 3") OR ("MARCAS CIP".RUN_CIP_TANQUE_4 AND NOT "DETECTOR FLUJO RET_L1" AND NOT "NIVEL MINIMO TQ 4") OR ("MARCAS CIP".RUN_CIP_TQ_21_S_LACTOSA AND NOT "DETECTOR FLUJO RET_L1" AND (NOT "LSL_TQ_21" OR "SIEMPRE_ON"))),
          operand := "Tag_773");
END_REGION

REGION Network 64: FIN DE CICLO
